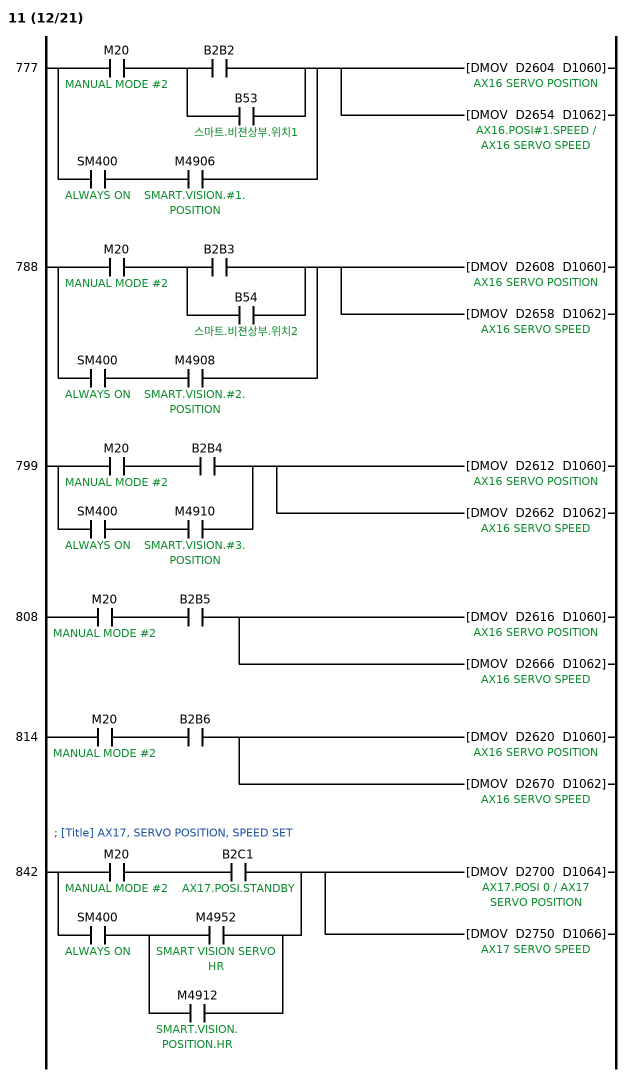
777   LD      M20  ; MANUAL MODE #2
      LD      B2B2
      OR      B53  ; 스마트.비젼상부.위치1
      ANB
      LD      SM400  ; ALWAYS ON
      AND     M4906  ; SMART.VISION.#1.POSITION
      ORB
      DMOV    D2604 D1060
      DMOV    D2654 D1062  ; AX16.POSI#1.SPEED
788   LD      M20  ; MANUAL MODE #2
      LD      B2B3
      OR      B54  ; 스마트.비젼상부.위치2
      ANB
      LD      SM400  ; ALWAYS ON
      AND     M4908  ; SMART.VISION.#2.POSITION
      ORB
      DMOV    D2608 D1060
      DMOV    D2658 D1062
799   LD      M20  ; MANUAL MODE #2
      AND     B2B4
      LD      SM400  ; ALWAYS ON
      AND     M4910  ; SMART.VISION.#3.POSITION
      ORB
      DMOV    D2612 D1060
      DMOV    D2662 D1062
808   LD      M20  ; MANUAL MODE #2
      AND     B2B5
      DMOV    D2616 D1060
      DMOV    D2666 D1062
814   LD      M20  ; MANUAL MODE #2
      AND     B2B6
      DMOV    D2620 D1060
      DMOV    D2670 D1062
; [Title] AX17, SERVO POSITION, SPEED SET
842   LD      M20  ; MANUAL MODE #2
      AND     B2C1  ; AX17.POSI.STANDBY
      LD      SM400  ; ALWAYS ON
      LD      M4952  ; SMART VISION SERVO HR
      OR      M4912  ; SMART.VISION.POSITION.HR
      ANB
      ORB
      DMOV    D2700 D1064  ; AX17.POSI 0
      DMOV    D2750 D1066
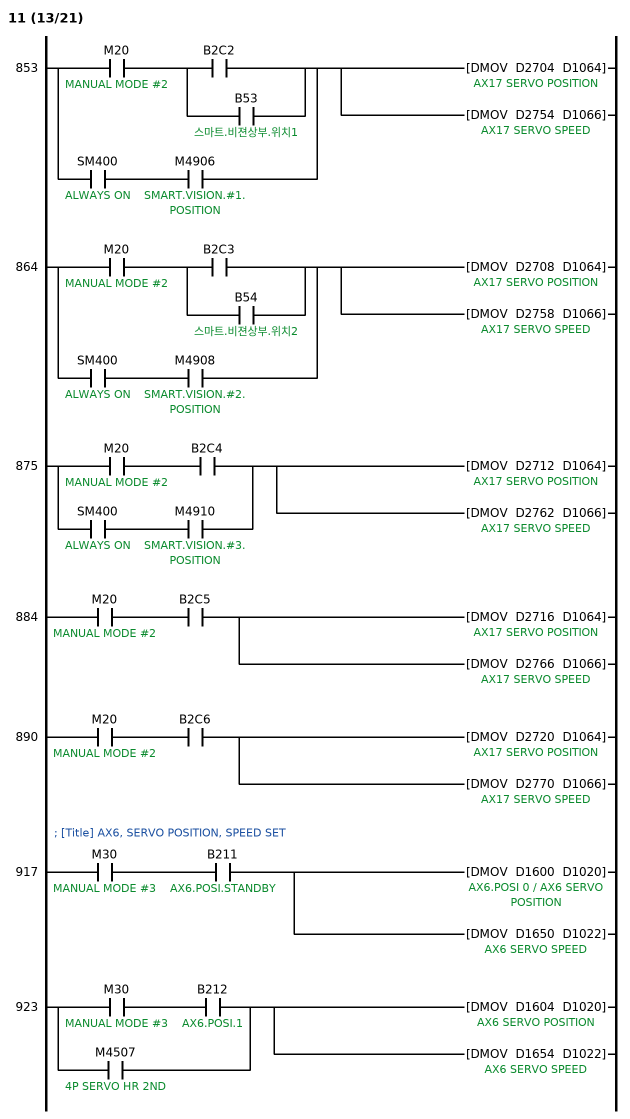
853   LD      M20  ; MANUAL MODE #2
      LD      B2C2
      OR      B53  ; 스마트.비젼상부.위치1
      ANB
      LD      SM400  ; ALWAYS ON
      AND     M4906  ; SMART.VISION.#1.POSITION
      ORB
      DMOV    D2704 D1064
      DMOV    D2754 D1066
864   LD      M20  ; MANUAL MODE #2
      LD      B2C3
      OR      B54  ; 스마트.비젼상부.위치2
      ANB
      LD      SM400  ; ALWAYS ON
      AND     M4908  ; SMART.VISION.#2.POSITION
      ORB
      DMOV    D2708 D1064
      DMOV    D2758 D1066
875   LD      M20  ; MANUAL MODE #2
      AND     B2C4
      LD      SM400  ; ALWAYS ON
      AND     M4910  ; SMART.VISION.#3.POSITION
      ORB
      DMOV    D2712 D1064
      DMOV    D2762 D1066
884   LD      M20  ; MANUAL MODE #2
      AND     B2C5
      DMOV    D2716 D1064
      DMOV    D2766 D1066
890   LD      M20  ; MANUAL MODE #2
      AND     B2C6
      DMOV    D2720 D1064
      DMOV    D2770 D1066
; [Title] AX6, SERVO POSITION, SPEED SET
917   LD      M30  ; MANUAL MODE #3
      AND     B211  ; AX6.POSI.STANDBY
      DMOV    D1600 D1020  ; AX6.POSI 0
      DMOV    D1650 D1022
923   LD      M30  ; MANUAL MODE #3
      AND     B212  ; AX6.POSI.1
      OR      M4507  ; 4P SERVO HR 2ND
      DMOV    D1604 D1020
      DMOV    D1654 D1022
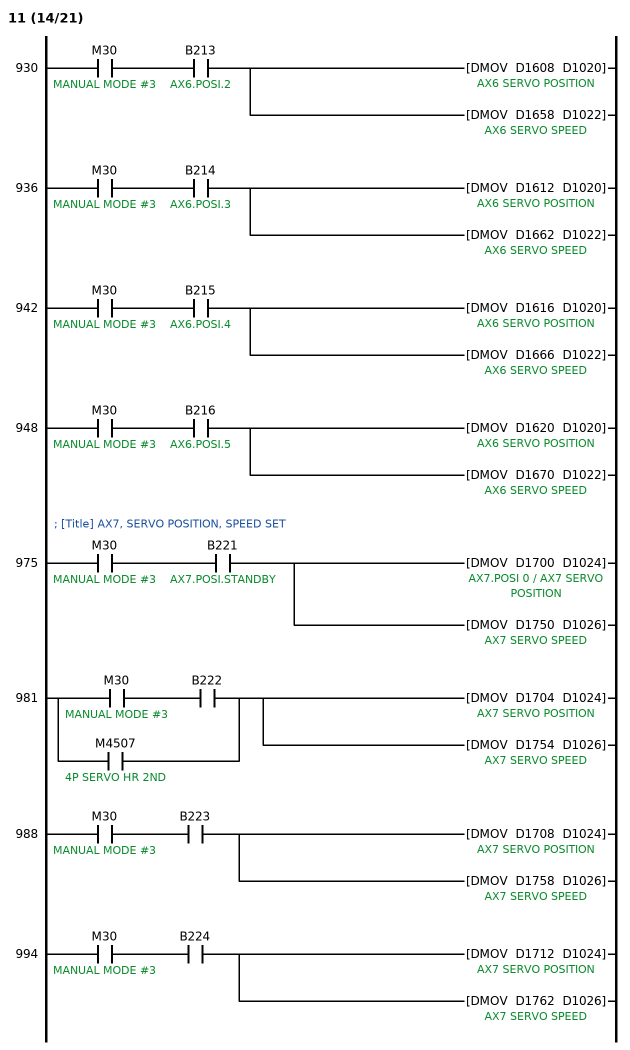
930   LD      M30  ; MANUAL MODE #3
      AND     B213  ; AX6.POSI.2
      DMOV    D1608 D1020
      DMOV    D1658 D1022
936   LD      M30  ; MANUAL MODE #3
      AND     B214  ; AX6.POSI.3
      DMOV    D1612 D1020
      DMOV    D1662 D1022
942   LD      M30  ; MANUAL MODE #3
      AND     B215  ; AX6.POSI.4
      DMOV    D1616 D1020
      DMOV    D1666 D1022
948   LD      M30  ; MANUAL MODE #3
      AND     B216  ; AX6.POSI.5
      DMOV    D1620 D1020
      DMOV    D1670 D1022
; [Title] AX7, SERVO POSITION, SPEED SET
975   LD      M30  ; MANUAL MODE #3
      AND     B221  ; AX7.POSI.STANDBY
      DMOV    D1700 D1024  ; AX7.POSI 0
      DMOV    D1750 D1026
981   LD      M30  ; MANUAL MODE #3
      AND     B222
      OR      M4507  ; 4P SERVO HR 2ND
      DMOV    D1704 D1024
      DMOV    D1754 D1026
988   LD      M30  ; MANUAL MODE #3
      AND     B223
      DMOV    D1708 D1024
      DMOV    D1758 D1026
994   LD      M30  ; MANUAL MODE #3
      AND     B224
      DMOV    D1712 D1024
      DMOV    D1762 D1026
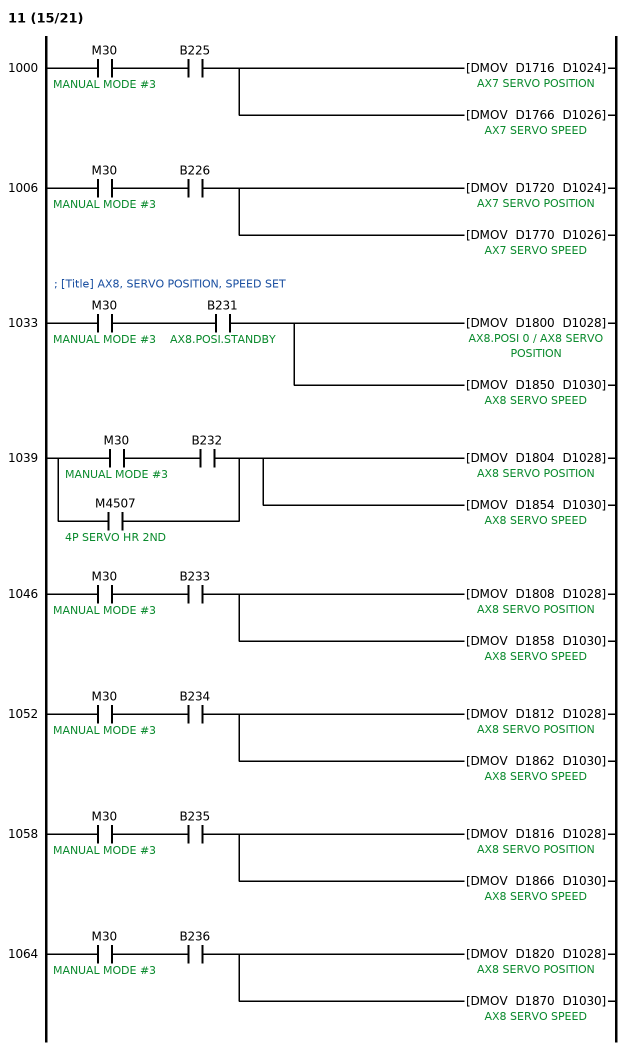
1000  LD      M30  ; MANUAL MODE #3
      AND     B225
      DMOV    D1716 D1024
      DMOV    D1766 D1026
1006  LD      M30  ; MANUAL MODE #3
      AND     B226
      DMOV    D1720 D1024
      DMOV    D1770 D1026
; [Title] AX8, SERVO POSITION, SPEED SET
1033  LD      M30  ; MANUAL MODE #3
      AND     B231  ; AX8.POSI.STANDBY
      DMOV    D1800 D1028  ; AX8.POSI 0
      DMOV    D1850 D1030
1039  LD      M30  ; MANUAL MODE #3
      AND     B232
      OR      M4507  ; 4P SERVO HR 2ND
      DMOV    D1804 D1028
      DMOV    D1854 D1030
1046  LD      M30  ; MANUAL MODE #3
      AND     B233
      DMOV    D1808 D1028
      DMOV    D1858 D1030
1052  LD      M30  ; MANUAL MODE #3
      AND     B234
      DMOV    D1812 D1028
      DMOV    D1862 D1030
1058  LD      M30  ; MANUAL MODE #3
      AND     B235
      DMOV    D1816 D1028
      DMOV    D1866 D1030
1064  LD      M30  ; MANUAL MODE #3
      AND     B236
      DMOV    D1820 D1028
      DMOV    D1870 D1030
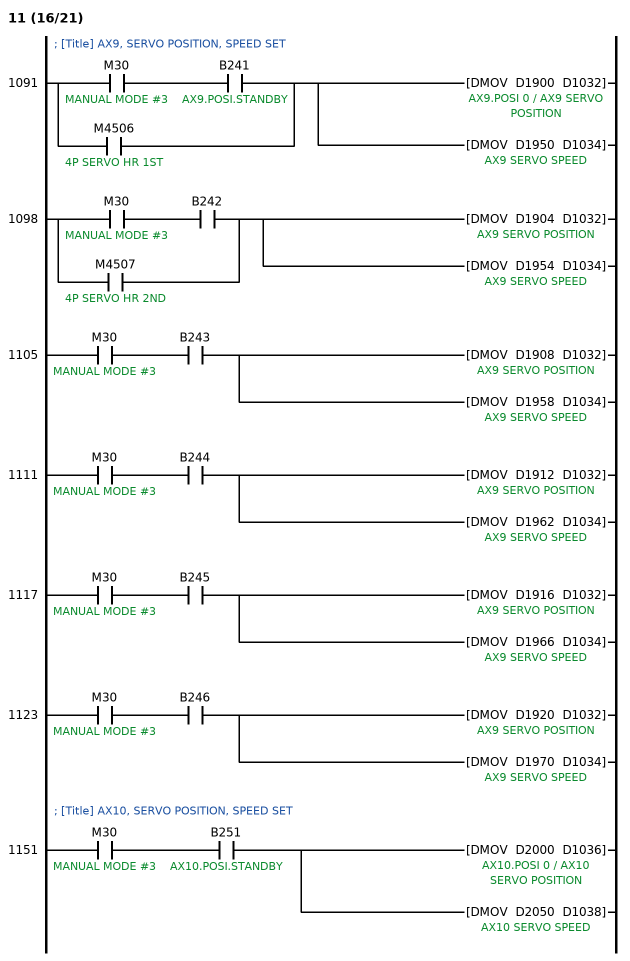
; [Title] AX9, SERVO POSITION, SPEED SET
1091  LD      M30  ; MANUAL MODE #3
      AND     B241  ; AX9.POSI.STANDBY
      OR      M4506  ; 4P SERVO HR 1ST
      DMOV    D1900 D1032  ; AX9.POSI 0
      DMOV    D1950 D1034
1098  LD      M30  ; MANUAL MODE #3
      AND     B242
      OR      M4507  ; 4P SERVO HR 2ND
      DMOV    D1904 D1032
      DMOV    D1954 D1034
1105  LD      M30  ; MANUAL MODE #3
      AND     B243
      DMOV    D1908 D1032
      DMOV    D1958 D1034
1111  LD      M30  ; MANUAL MODE #3
      AND     B244
      DMOV    D1912 D1032
      DMOV    D1962 D1034
1117  LD      M30  ; MANUAL MODE #3
      AND     B245
      DMOV    D1916 D1032
      DMOV    D1966 D1034
1123  LD      M30  ; MANUAL MODE #3
      AND     B246
      DMOV    D1920 D1032
      DMOV    D1970 D1034
; [Title] AX10, SERVO POSITION, SPEED SET
1151  LD      M30  ; MANUAL MODE #3
      AND     B251  ; AX10.POSI.STANDBY
      DMOV    D2000 D1036  ; AX10.POSI 0
      DMOV    D2050 D1038
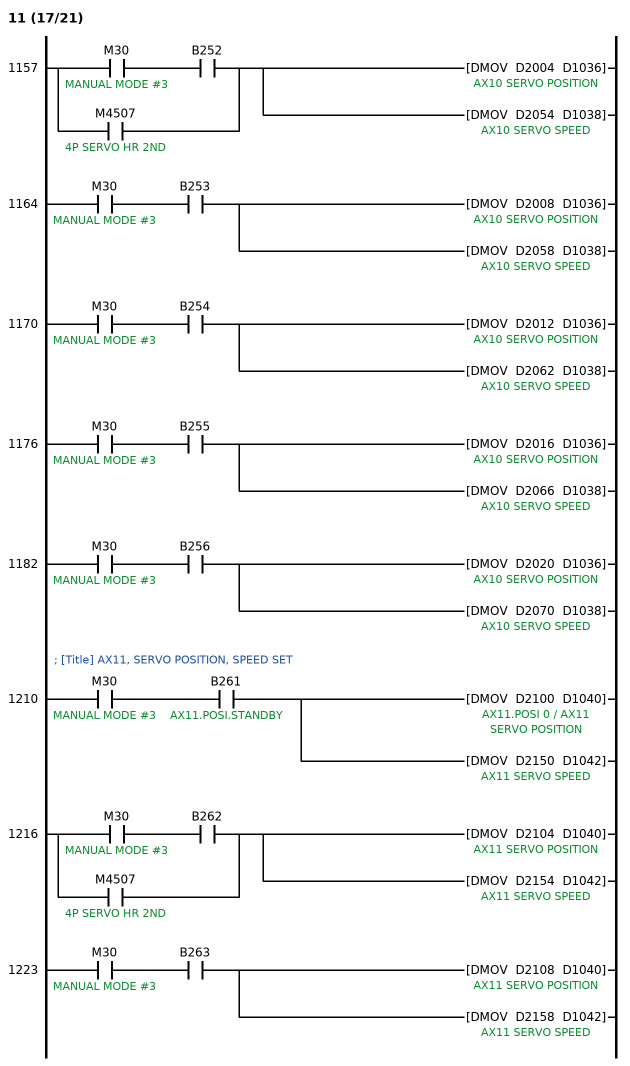
1157  LD      M30  ; MANUAL MODE #3
      AND     B252
      OR      M4507  ; 4P SERVO HR 2ND
      DMOV    D2004 D1036
      DMOV    D2054 D1038
1164  LD      M30  ; MANUAL MODE #3
      AND     B253
      DMOV    D2008 D1036
      DMOV    D2058 D1038
1170  LD      M30  ; MANUAL MODE #3
      AND     B254
      DMOV    D2012 D1036
      DMOV    D2062 D1038
1176  LD      M30  ; MANUAL MODE #3
      AND     B255
      DMOV    D2016 D1036
      DMOV    D2066 D1038
1182  LD      M30  ; MANUAL MODE #3
      AND     B256
      DMOV    D2020 D1036
      DMOV    D2070 D1038
; [Title] AX11, SERVO POSITION, SPEED SET
1210  LD      M30  ; MANUAL MODE #3
      AND     B261  ; AX11.POSI.STANDBY
      DMOV    D2100 D1040  ; AX11.POSI 0
      DMOV    D2150 D1042
1216  LD      M30  ; MANUAL MODE #3
      AND     B262
      OR      M4507  ; 4P SERVO HR 2ND
      DMOV    D2104 D1040
      DMOV    D2154 D1042
1223  LD      M30  ; MANUAL MODE #3
      AND     B263
      DMOV    D2108 D1040
      DMOV    D2158 D1042
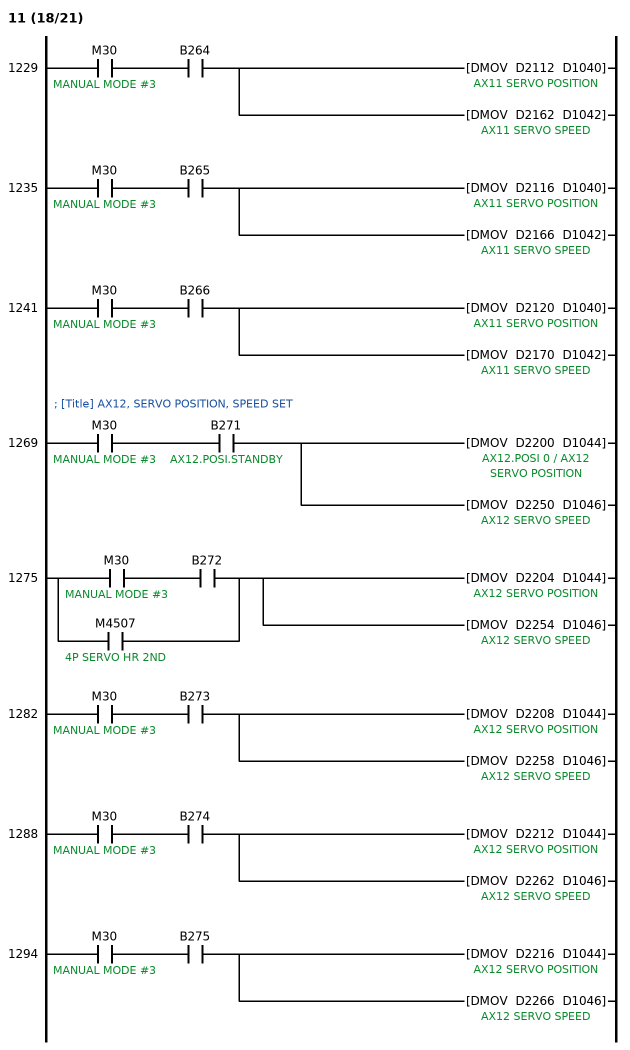
1229  LD      M30  ; MANUAL MODE #3
      AND     B264
      DMOV    D2112 D1040
      DMOV    D2162 D1042
1235  LD      M30  ; MANUAL MODE #3
      AND     B265
      DMOV    D2116 D1040
      DMOV    D2166 D1042
1241  LD      M30  ; MANUAL MODE #3
      AND     B266
      DMOV    D2120 D1040
      DMOV    D2170 D1042
; [Title] AX12, SERVO POSITION, SPEED SET
1269  LD      M30  ; MANUAL MODE #3
      AND     B271  ; AX12.POSI.STANDBY
      DMOV    D2200 D1044  ; AX12.POSI 0
      DMOV    D2250 D1046
1275  LD      M30  ; MANUAL MODE #3
      AND     B272
      OR      M4507  ; 4P SERVO HR 2ND
      DMOV    D2204 D1044
      DMOV    D2254 D1046
1282  LD      M30  ; MANUAL MODE #3
      AND     B273
      DMOV    D2208 D1044
      DMOV    D2258 D1046
1288  LD      M30  ; MANUAL MODE #3
      AND     B274
      DMOV    D2212 D1044
      DMOV    D2262 D1046
1294  LD      M30  ; MANUAL MODE #3
      AND     B275
      DMOV    D2216 D1044
      DMOV    D2266 D1046
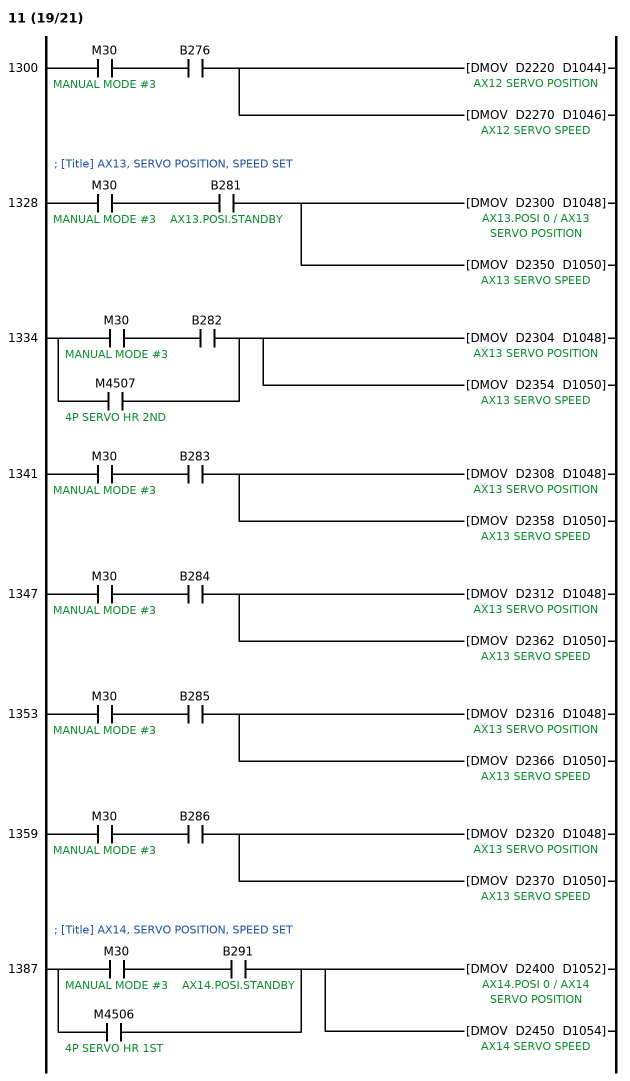
1300  LD      M30  ; MANUAL MODE #3
      AND     B276
      DMOV    D2220 D1044
      DMOV    D2270 D1046
; [Title] AX13, SERVO POSITION, SPEED SET
1328  LD      M30  ; MANUAL MODE #3
      AND     B281  ; AX13.POSI.STANDBY
      DMOV    D2300 D1048  ; AX13.POSI 0
      DMOV    D2350 D1050
1334  LD      M30  ; MANUAL MODE #3
      AND     B282
      OR      M4507  ; 4P SERVO HR 2ND
      DMOV    D2304 D1048
      DMOV    D2354 D1050
1341  LD      M30  ; MANUAL MODE #3
      AND     B283
      DMOV    D2308 D1048
      DMOV    D2358 D1050
1347  LD      M30  ; MANUAL MODE #3
      AND     B284
      DMOV    D2312 D1048
      DMOV    D2362 D1050
1353  LD      M30  ; MANUAL MODE #3
      AND     B285
      DMOV    D2316 D1048
      DMOV    D2366 D1050
1359  LD      M30  ; MANUAL MODE #3
      AND     B286
      DMOV    D2320 D1048
      DMOV    D2370 D1050
; [Title] AX14, SERVO POSITION, SPEED SET
1387  LD      M30  ; MANUAL MODE #3
      AND     B291  ; AX14.POSI.STANDBY
      OR      M4506  ; 4P SERVO HR 1ST
      DMOV    D2400 D1052  ; AX14.POSI 0
      DMOV    D2450 D1054
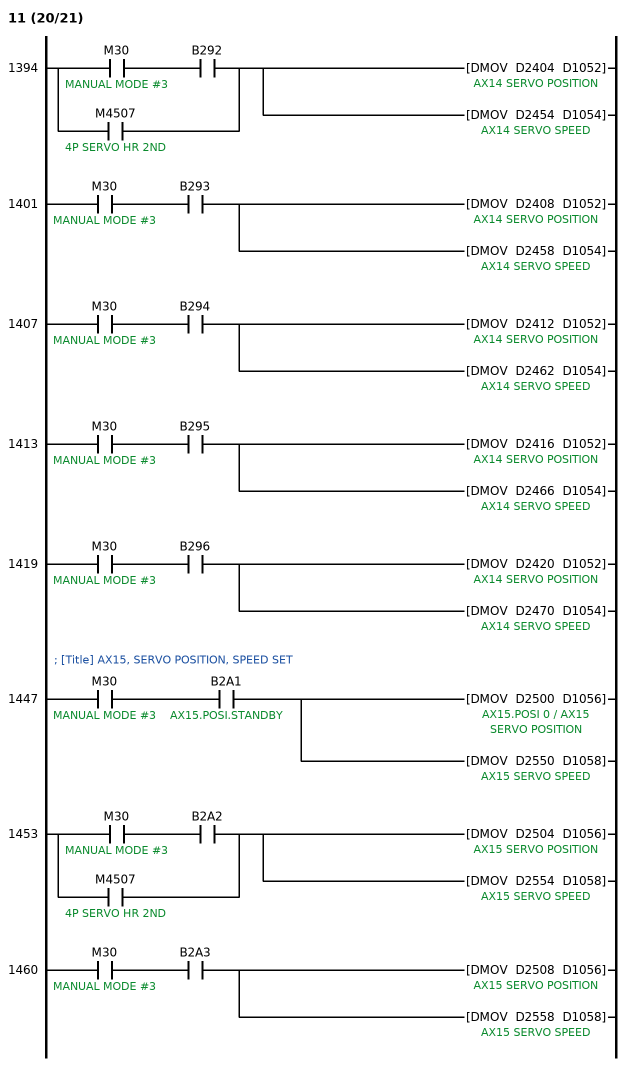
1394  LD      M30  ; MANUAL MODE #3
      AND     B292
      OR      M4507  ; 4P SERVO HR 2ND
      DMOV    D2404 D1052
      DMOV    D2454 D1054
1401  LD      M30  ; MANUAL MODE #3
      AND     B293
      DMOV    D2408 D1052
      DMOV    D2458 D1054
1407  LD      M30  ; MANUAL MODE #3
      AND     B294
      DMOV    D2412 D1052
      DMOV    D2462 D1054
1413  LD      M30  ; MANUAL MODE #3
      AND     B295
      DMOV    D2416 D1052
      DMOV    D2466 D1054
1419  LD      M30  ; MANUAL MODE #3
      AND     B296
      DMOV    D2420 D1052
      DMOV    D2470 D1054
; [Title] AX15, SERVO POSITION, SPEED SET
1447  LD      M30  ; MANUAL MODE #3
      AND     B2A1  ; AX15.POSI.STANDBY
      DMOV    D2500 D1056  ; AX15.POSI 0
      DMOV    D2550 D1058
1453  LD      M30  ; MANUAL MODE #3
      AND     B2A2
      OR      M4507  ; 4P SERVO HR 2ND
      DMOV    D2504 D1056
      DMOV    D2554 D1058
1460  LD      M30  ; MANUAL MODE #3
      AND     B2A3
      DMOV    D2508 D1056
      DMOV    D2558 D1058
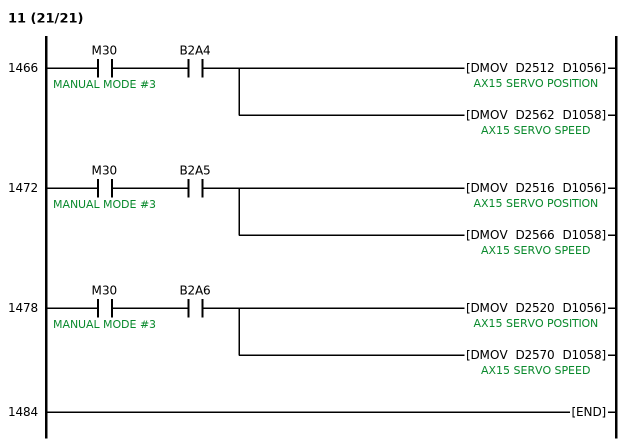
1466  LD      M30  ; MANUAL MODE #3
      AND     B2A4
      DMOV    D2512 D1056
      DMOV    D2562 D1058
1472  LD      M30  ; MANUAL MODE #3
      AND     B2A5
      DMOV    D2516 D1056
      DMOV    D2566 D1058
1478  LD      M30  ; MANUAL MODE #3
      AND     B2A6
      DMOV    D2520 D1056
      DMOV    D2570 D1058
1484  END
END_PROGRAM

PROGRAM 12  // SERVO DATA (2)
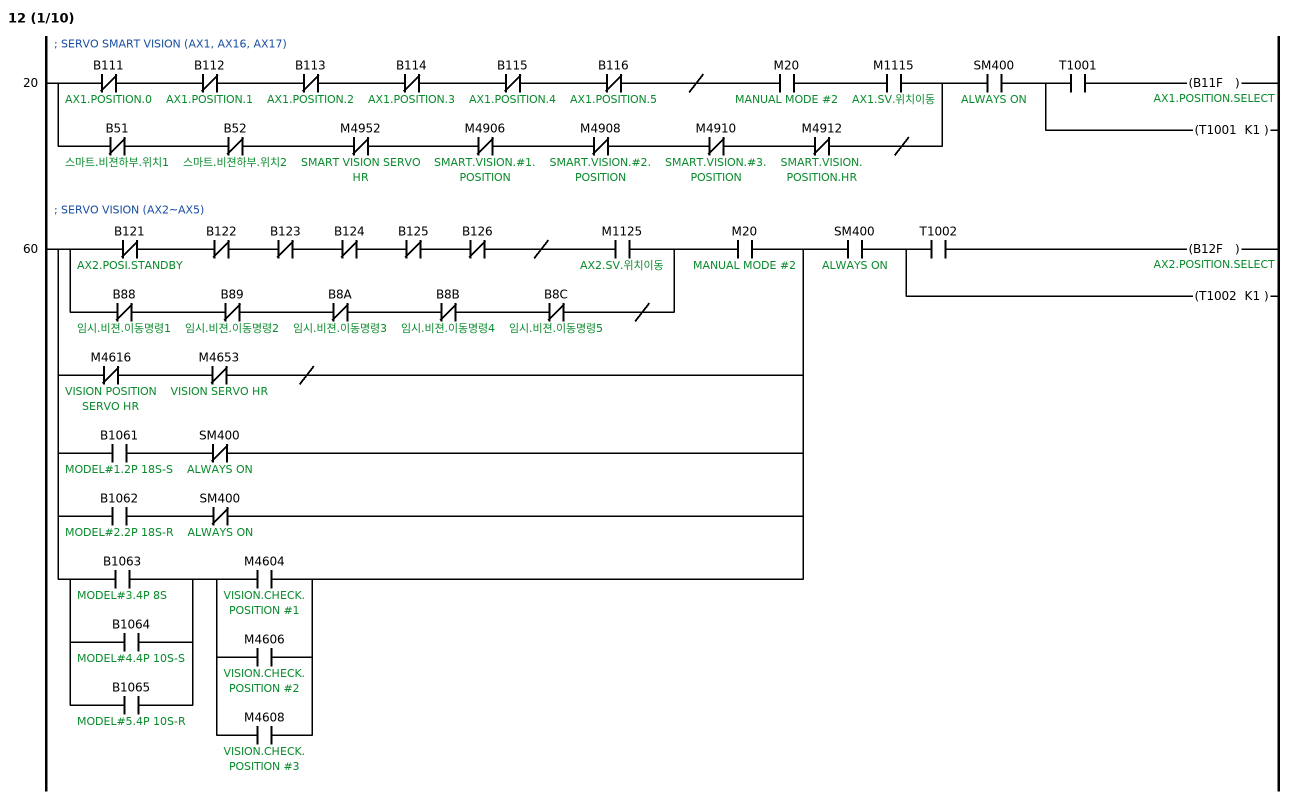
; SERVO SMART VISION (AX1, AX16, AX17)
20    LDI     B111  ; AX1.POSITION.0
      ANI     B112  ; AX1.POSITION.1
      ANI     B113  ; AX1.POSITION.2
      ANI     B114  ; AX1.POSITION.3
      ANI     B115  ; AX1.POSITION.4
      ANI     B116  ; AX1.POSITION.5
      INV
      AND     M20  ; MANUAL MODE #2
      AND     M1115  ; AX1.SV.위치이동
      LDI     B51  ; 스마트.비젼하부.위치1
      ANI     B52  ; 스마트.비젼하부.위치2
      ANI     M4952  ; SMART VISION SERVO HR
      ANI     M4906  ; SMART.VISION.#1.POSITION
      ANI     M4908  ; SMART.VISION.#2.POSITION
      ANI     M4910  ; SMART.VISION.#3.POSITION
      ANI     M4912  ; SMART.VISION.POSITION.HR
      INV
      ORB
      AND     SM400  ; ALWAYS ON
      MPS
      AND     T1001
      OUT     B11F  ; AX1.POSITION.SELECT
      MPP
      OUT     T1001 K1
; SERVO VISION (AX2~AX5)
60    LDI     B121  ; AX2.POSI.STANDBY
      ANI     B122
      ANI     B123
      ANI     B124
      ANI     B125
      ANI     B126
      INV
      AND     M1125  ; AX2.SV.위치이동
      LDI     B88  ; 임시.비젼.이동명령1
      ANI     B89  ; 임시.비젼.이동명령2
      ANI     B8A  ; 임시.비젼.이동명령3
      ANI     B8B  ; 임시.비젼.이동명령4
      ANI     B8C  ; 임시.비젼.이동명령5
      INV
      ORB
      AND     M20  ; MANUAL MODE #2
      LDI     M4616  ; VISION POSITION SERVO HR
      ANI     M4653  ; VISION SERVO HR
      INV
      ORB
      LD      B1061  ; MODEL#1.2P 18S-S
      ANI     SM400  ; ALWAYS ON
      ORB
      LD      B1062  ; MODEL#2.2P 18S-R
      ANI     SM400  ; ALWAYS ON
      ORB
      LD      B1063  ; MODEL#3.4P 8S
      OR      B1064  ; MODEL#4.4P 10S-S
      OR      B1065  ; MODEL#5.4P 10S-R
      LD      M4604  ; VISION.CHECK.POSITION #1
      OR      M4606  ; VISION.CHECK.POSITION #2
      OR      M4608  ; VISION.CHECK.POSITION #3
      ANB
      ORB
      AND     SM400  ; ALWAYS ON
      MPS
      AND     T1002
      OUT     B12F  ; AX2.POSITION.SELECT
      MPP
      OUT     T1002 K1
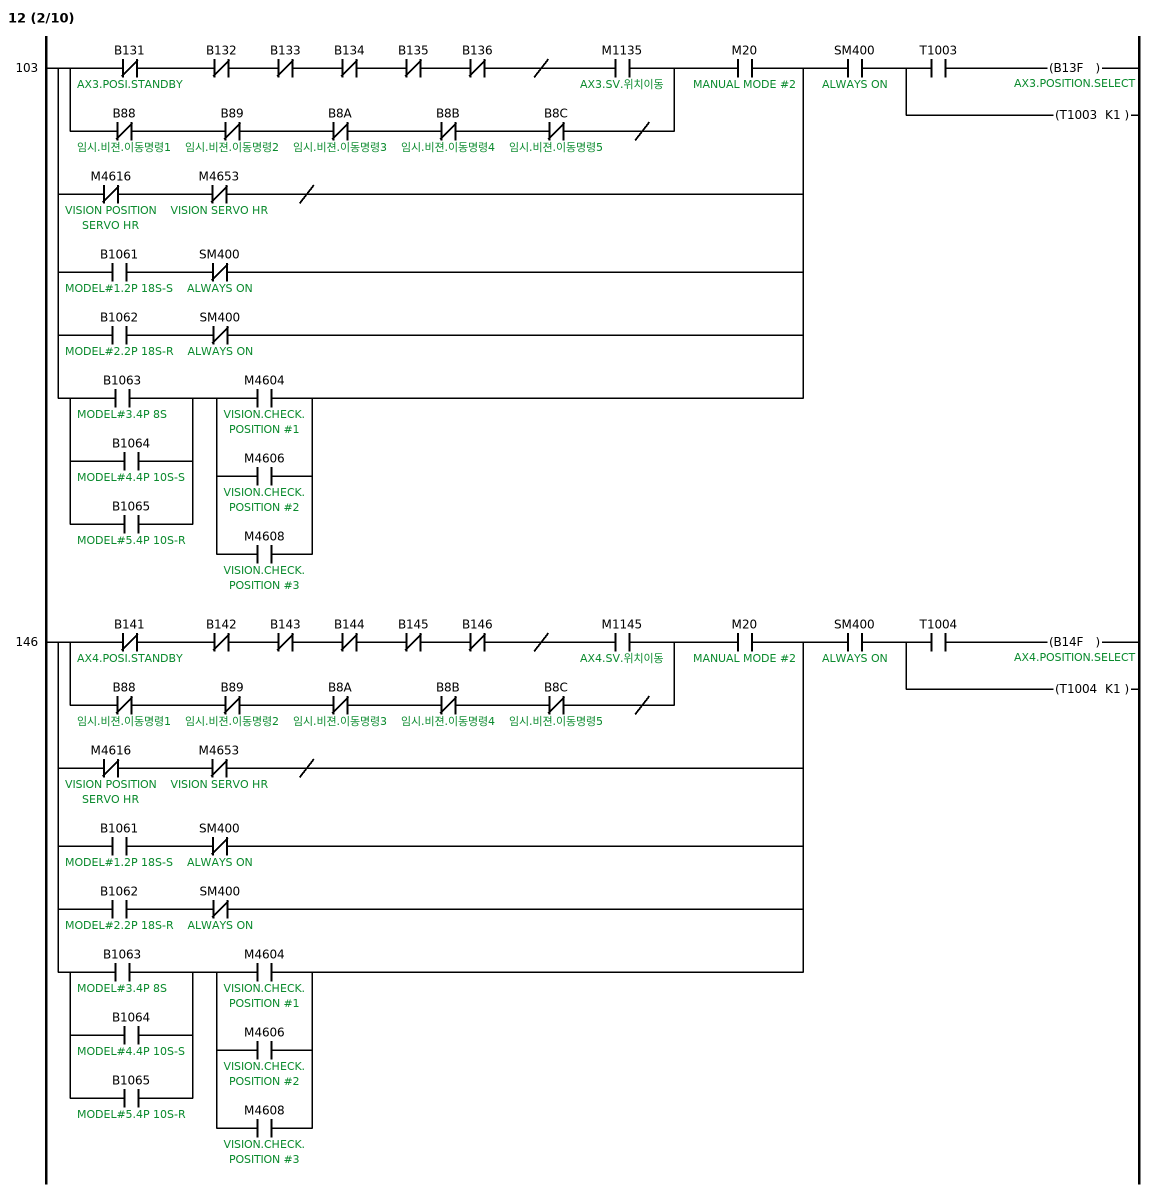
103   LDI     B131  ; AX3.POSI.STANDBY
      ANI     B132
      ANI     B133
      ANI     B134
      ANI     B135
      ANI     B136
      INV
      AND     M1135  ; AX3.SV.위치이동
      LDI     B88  ; 임시.비젼.이동명령1
      ANI     B89  ; 임시.비젼.이동명령2
      ANI     B8A  ; 임시.비젼.이동명령3
      ANI     B8B  ; 임시.비젼.이동명령4
      ANI     B8C  ; 임시.비젼.이동명령5
      INV
      ORB
      AND     M20  ; MANUAL MODE #2
      LDI     M4616  ; VISION POSITION SERVO HR
      ANI     M4653  ; VISION SERVO HR
      INV
      ORB
      LD      B1061  ; MODEL#1.2P 18S-S
      ANI     SM400  ; ALWAYS ON
      ORB
      LD      B1062  ; MODEL#2.2P 18S-R
      ANI     SM400  ; ALWAYS ON
      ORB
      LD      B1063  ; MODEL#3.4P 8S
      OR      B1064  ; MODEL#4.4P 10S-S
      OR      B1065  ; MODEL#5.4P 10S-R
      LD      M4604  ; VISION.CHECK.POSITION #1
      OR      M4606  ; VISION.CHECK.POSITION #2
      OR      M4608  ; VISION.CHECK.POSITION #3
      ANB
      ORB
      AND     SM400  ; ALWAYS ON
      MPS
      AND     T1003
      OUT     B13F  ; AX3.POSITION.SELECT
      MPP
      OUT     T1003 K1
146   LDI     B141  ; AX4.POSI.STANDBY
      ANI     B142
      ANI     B143
      ANI     B144
      ANI     B145
      ANI     B146
      INV
      AND     M1145  ; AX4.SV.위치이동
      LDI     B88  ; 임시.비젼.이동명령1
      ANI     B89  ; 임시.비젼.이동명령2
      ANI     B8A  ; 임시.비젼.이동명령3
      ANI     B8B  ; 임시.비젼.이동명령4
      ANI     B8C  ; 임시.비젼.이동명령5
      INV
      ORB
      AND     M20  ; MANUAL MODE #2
      LDI     M4616  ; VISION POSITION SERVO HR
      ANI     M4653  ; VISION SERVO HR
      INV
      ORB
      LD      B1061  ; MODEL#1.2P 18S-S
      ANI     SM400  ; ALWAYS ON
      ORB
      LD      B1062  ; MODEL#2.2P 18S-R
      ANI     SM400  ; ALWAYS ON
      ORB
      LD      B1063  ; MODEL#3.4P 8S
      OR      B1064  ; MODEL#4.4P 10S-S
      OR      B1065  ; MODEL#5.4P 10S-R
      LD      M4604  ; VISION.CHECK.POSITION #1
      OR      M4606  ; VISION.CHECK.POSITION #2
      OR      M4608  ; VISION.CHECK.POSITION #3
      ANB
      ORB
      AND     SM400  ; ALWAYS ON
      MPS
      AND     T1004
      OUT     B14F  ; AX4.POSITION.SELECT
      MPP
      OUT     T1004 K1
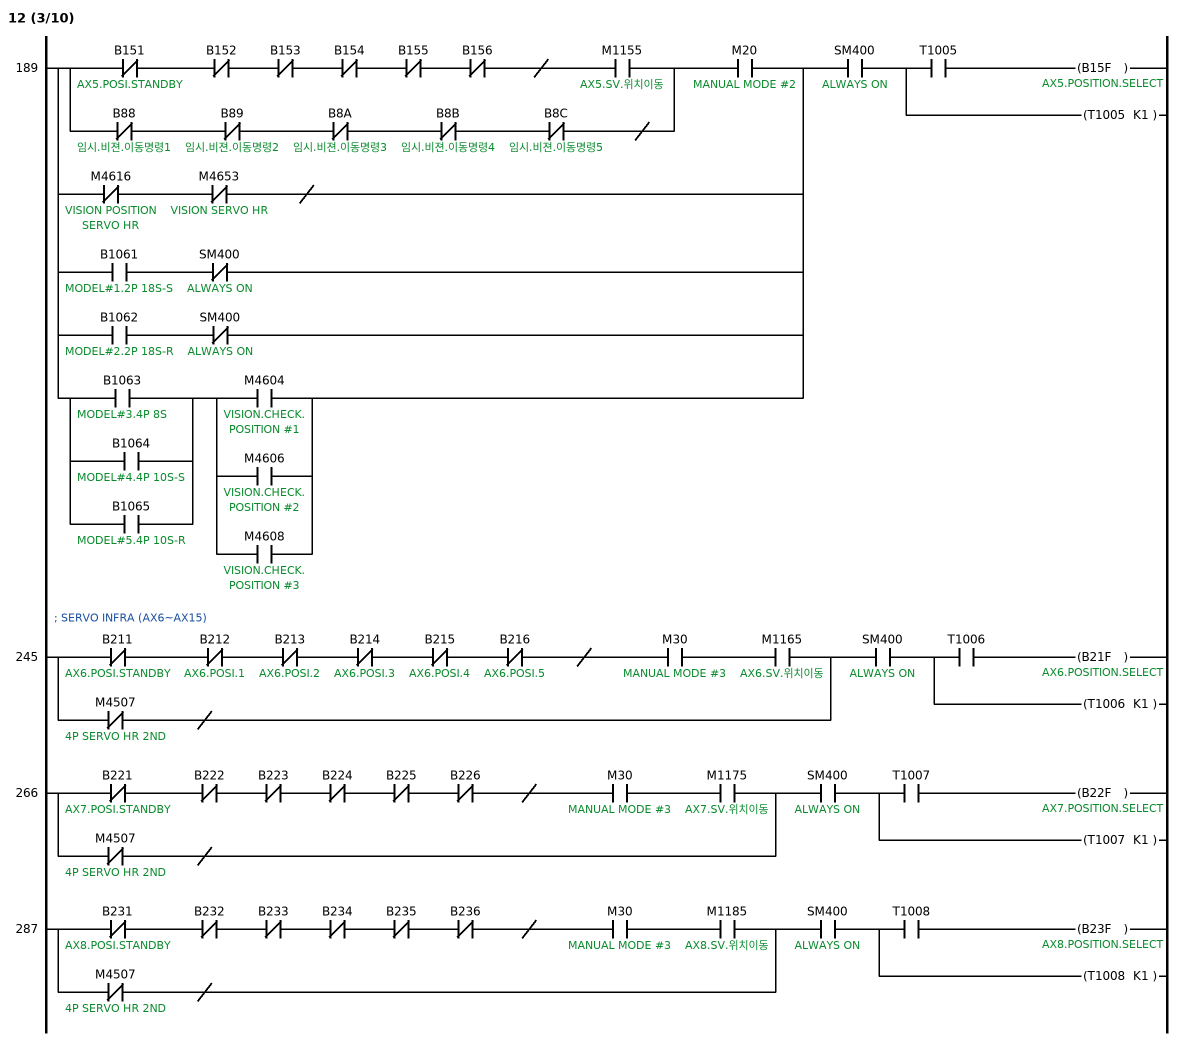
189   LDI     B151  ; AX5.POSI.STANDBY
      ANI     B152
      ANI     B153
      ANI     B154
      ANI     B155
      ANI     B156
      INV
      AND     M1155  ; AX5.SV.위치이동
      LDI     B88  ; 임시.비젼.이동명령1
      ANI     B89  ; 임시.비젼.이동명령2
      ANI     B8A  ; 임시.비젼.이동명령3
      ANI     B8B  ; 임시.비젼.이동명령4
      ANI     B8C  ; 임시.비젼.이동명령5
      INV
      ORB
      AND     M20  ; MANUAL MODE #2
      LDI     M4616  ; VISION POSITION SERVO HR
      ANI     M4653  ; VISION SERVO HR
      INV
      ORB
      LD      B1061  ; MODEL#1.2P 18S-S
      ANI     SM400  ; ALWAYS ON
      ORB
      LD      B1062  ; MODEL#2.2P 18S-R
      ANI     SM400  ; ALWAYS ON
      ORB
      LD      B1063  ; MODEL#3.4P 8S
      OR      B1064  ; MODEL#4.4P 10S-S
      OR      B1065  ; MODEL#5.4P 10S-R
      LD      M4604  ; VISION.CHECK.POSITION #1
      OR      M4606  ; VISION.CHECK.POSITION #2
      OR      M4608  ; VISION.CHECK.POSITION #3
      ANB
      ORB
      AND     SM400  ; ALWAYS ON
      MPS
      AND     T1005
      OUT     B15F  ; AX5.POSITION.SELECT
      MPP
      OUT     T1005 K1
; SERVO INFRA (AX6~AX15)
245   LDI     B211  ; AX6.POSI.STANDBY
      ANI     B212  ; AX6.POSI.1
      ANI     B213  ; AX6.POSI.2
      ANI     B214  ; AX6.POSI.3
      ANI     B215  ; AX6.POSI.4
      ANI     B216  ; AX6.POSI.5
      INV
      AND     M30  ; MANUAL MODE #3
      AND     M1165  ; AX6.SV.위치이동
      LDI     M4507  ; 4P SERVO HR 2ND
      INV
      ORB
      AND     SM400  ; ALWAYS ON
      MPS
      AND     T1006
      OUT     B21F  ; AX6.POSITION.SELECT
      MPP
      OUT     T1006 K1
266   LDI     B221  ; AX7.POSI.STANDBY
      ANI     B222
      ANI     B223
      ANI     B224
      ANI     B225
      ANI     B226
      INV
      AND     M30  ; MANUAL MODE #3
      AND     M1175  ; AX7.SV.위치이동
      LDI     M4507  ; 4P SERVO HR 2ND
      INV
      ORB
      AND     SM400  ; ALWAYS ON
      MPS
      AND     T1007
      OUT     B22F  ; AX7.POSITION.SELECT
      MPP
      OUT     T1007 K1
287   LDI     B231  ; AX8.POSI.STANDBY
      ANI     B232
      ANI     B233
      ANI     B234
      ANI     B235
      ANI     B236
      INV
      AND     M30  ; MANUAL MODE #3
      AND     M1185  ; AX8.SV.위치이동
      LDI     M4507  ; 4P SERVO HR 2ND
      INV
      ORB
      AND     SM400  ; ALWAYS ON
      MPS
      AND     T1008
      OUT     B23F  ; AX8.POSITION.SELECT
      MPP
      OUT     T1008 K1
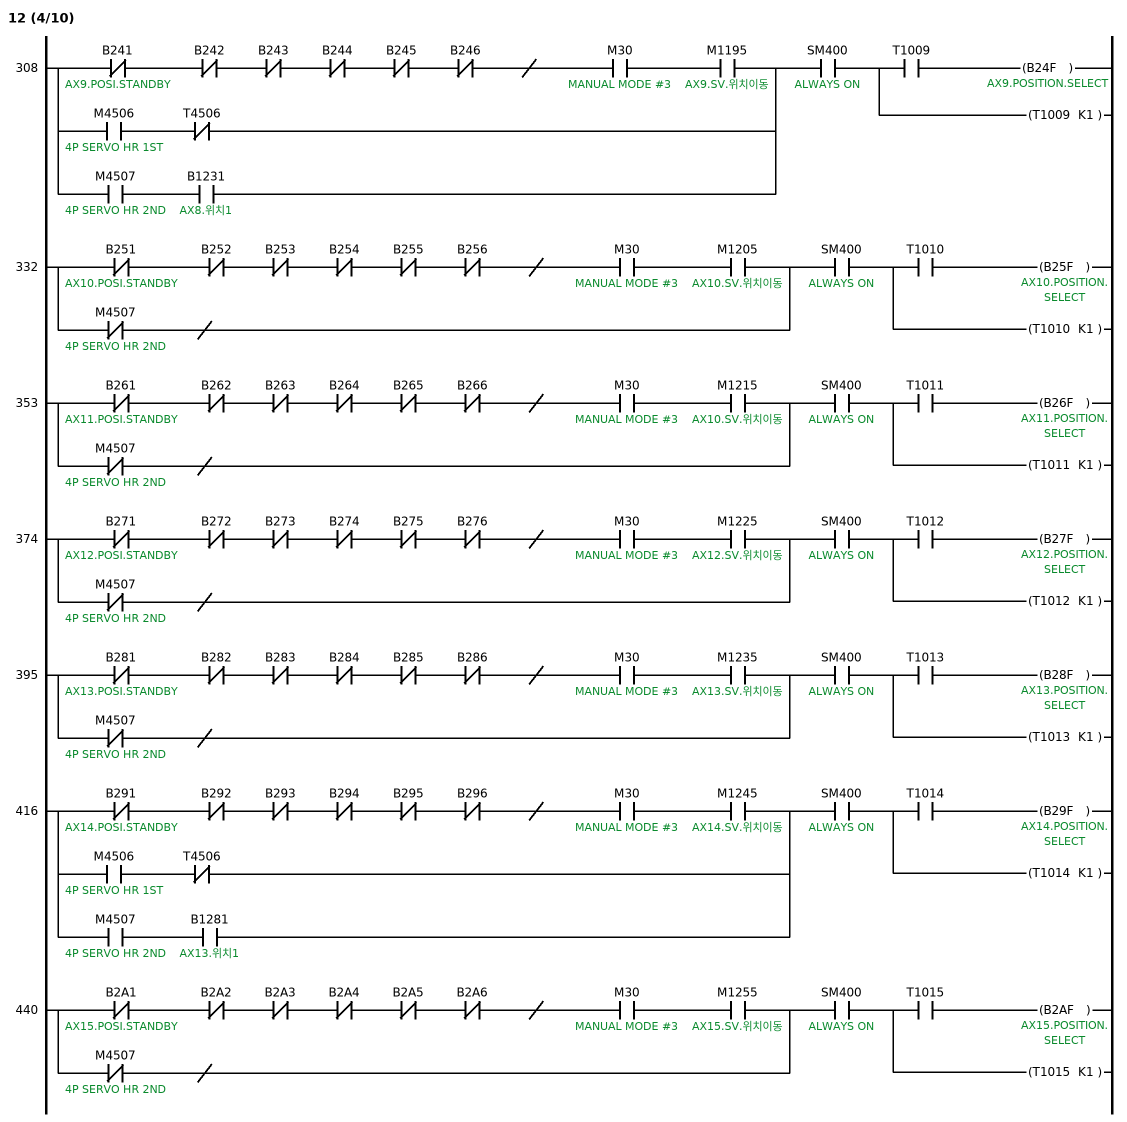
308   LDI     B241  ; AX9.POSI.STANDBY
      ANI     B242
      ANI     B243
      ANI     B244
      ANI     B245
      ANI     B246
      INV
      AND     M30  ; MANUAL MODE #3
      AND     M1195  ; AX9.SV.위치이동
      LD      M4506  ; 4P SERVO HR 1ST
      ANI     T4506
      ORB
      LD      M4507  ; 4P SERVO HR 2ND
      AND     B1231  ; AX8.위치1
      ORB
      AND     SM400  ; ALWAYS ON
      MPS
      AND     T1009
      OUT     B24F  ; AX9.POSITION.SELECT
      MPP
      OUT     T1009 K1
332   LDI     B251  ; AX10.POSI.STANDBY
      ANI     B252
      ANI     B253
      ANI     B254
      ANI     B255
      ANI     B256
      INV
      AND     M30  ; MANUAL MODE #3
      AND     M1205  ; AX10.SV.위치이동
      LDI     M4507  ; 4P SERVO HR 2ND
      INV
      ORB
      AND     SM400  ; ALWAYS ON
      MPS
      AND     T1010
      OUT     B25F  ; AX10.POSITION.SELECT
      MPP
      OUT     T1010 K1
353   LDI     B261  ; AX11.POSI.STANDBY
      ANI     B262
      ANI     B263
      ANI     B264
      ANI     B265
      ANI     B266
      INV
      AND     M30  ; MANUAL MODE #3
      AND     M1215  ; AX10.SV.위치이동
      LDI     M4507  ; 4P SERVO HR 2ND
      INV
      ORB
      AND     SM400  ; ALWAYS ON
      MPS
      AND     T1011
      OUT     B26F  ; AX11.POSITION.SELECT
      MPP
      OUT     T1011 K1
374   LDI     B271  ; AX12.POSI.STANDBY
      ANI     B272
      ANI     B273
      ANI     B274
      ANI     B275
      ANI     B276
      INV
      AND     M30  ; MANUAL MODE #3
      AND     M1225  ; AX12.SV.위치이동
      LDI     M4507  ; 4P SERVO HR 2ND
      INV
      ORB
      AND     SM400  ; ALWAYS ON
      MPS
      AND     T1012
      OUT     B27F  ; AX12.POSITION.SELECT
      MPP
      OUT     T1012 K1
395   LDI     B281  ; AX13.POSI.STANDBY
      ANI     B282
      ANI     B283
      ANI     B284
      ANI     B285
      ANI     B286
      INV
      AND     M30  ; MANUAL MODE #3
      AND     M1235  ; AX13.SV.위치이동
      LDI     M4507  ; 4P SERVO HR 2ND
      INV
      ORB
      AND     SM400  ; ALWAYS ON
      MPS
      AND     T1013
      OUT     B28F  ; AX13.POSITION.SELECT
      MPP
      OUT     T1013 K1
416   LDI     B291  ; AX14.POSI.STANDBY
      ANI     B292
      ANI     B293
      ANI     B294
      ANI     B295
      ANI     B296
      INV
      AND     M30  ; MANUAL MODE #3
      AND     M1245  ; AX14.SV.위치이동
      LD      M4506  ; 4P SERVO HR 1ST
      ANI     T4506
      ORB
      LD      M4507  ; 4P SERVO HR 2ND
      AND     B1281  ; AX13.위치1
      ORB
      AND     SM400  ; ALWAYS ON
      MPS
      AND     T1014
      OUT     B29F  ; AX14.POSITION.SELECT
      MPP
      OUT     T1014 K1
440   LDI     B2A1  ; AX15.POSI.STANDBY
      ANI     B2A2
      ANI     B2A3
      ANI     B2A4
      ANI     B2A5
      ANI     B2A6
      INV
      AND     M30  ; MANUAL MODE #3
      AND     M1255  ; AX15.SV.위치이동
      LDI     M4507  ; 4P SERVO HR 2ND
      INV
      ORB
      AND     SM400  ; ALWAYS ON
      MPS
      AND     T1015
      OUT     B2AF  ; AX15.POSITION.SELECT
      MPP
      OUT     T1015 K1
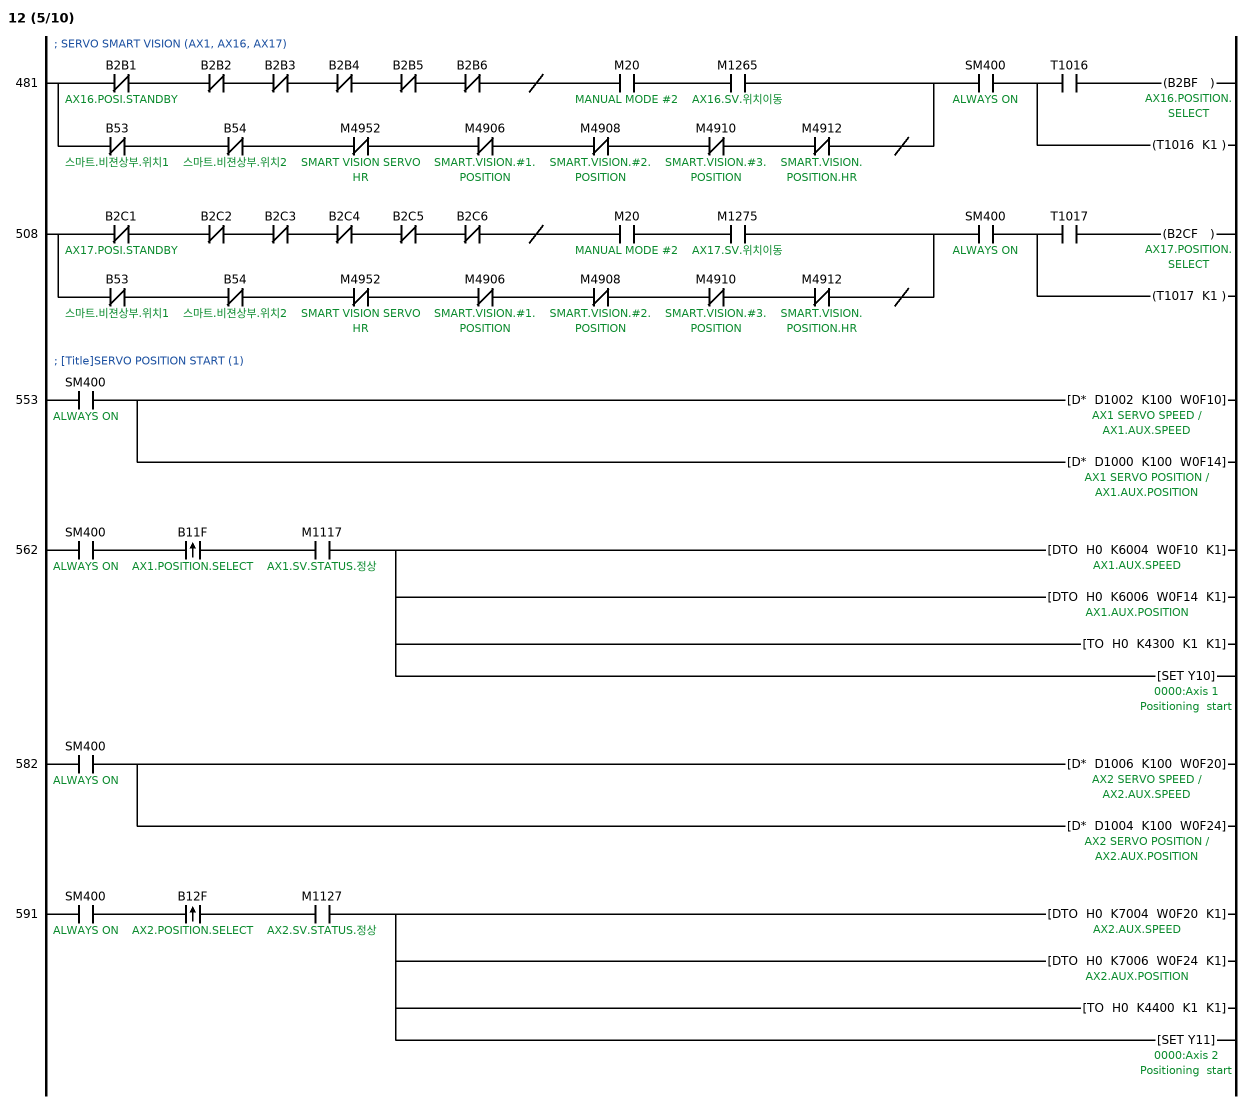
; SERVO SMART VISION (AX1, AX16, AX17)
481   LDI     B2B1  ; AX16.POSI.STANDBY
      ANI     B2B2
      ANI     B2B3
      ANI     B2B4
      ANI     B2B5
      ANI     B2B6
      INV
      AND     M20  ; MANUAL MODE #2
      AND     M1265  ; AX16.SV.위치이동
      LDI     B53  ; 스마트.비젼상부.위치1
      ANI     B54  ; 스마트.비젼상부.위치2
      ANI     M4952  ; SMART VISION SERVO HR
      ANI     M4906  ; SMART.VISION.#1.POSITION
      ANI     M4908  ; SMART.VISION.#2.POSITION
      ANI     M4910  ; SMART.VISION.#3.POSITION
      ANI     M4912  ; SMART.VISION.POSITION.HR
      INV
      ORB
      AND     SM400  ; ALWAYS ON
      MPS
      AND     T1016
      OUT     B2BF  ; AX16.POSITION.SELECT
      MPP
      OUT     T1016 K1
508   LDI     B2C1  ; AX17.POSI.STANDBY
      ANI     B2C2
      ANI     B2C3
      ANI     B2C4
      ANI     B2C5
      ANI     B2C6
      INV
      AND     M20  ; MANUAL MODE #2
      AND     M1275  ; AX17.SV.위치이동
      LDI     B53  ; 스마트.비젼상부.위치1
      ANI     B54  ; 스마트.비젼상부.위치2
      ANI     M4952  ; SMART VISION SERVO HR
      ANI     M4906  ; SMART.VISION.#1.POSITION
      ANI     M4908  ; SMART.VISION.#2.POSITION
      ANI     M4910  ; SMART.VISION.#3.POSITION
      ANI     M4912  ; SMART.VISION.POSITION.HR
      INV
      ORB
      AND     SM400  ; ALWAYS ON
      MPS
      AND     T1017
      OUT     B2CF  ; AX17.POSITION.SELECT
      MPP
      OUT     T1017 K1
; [Title]SERVO POSITION START (1)
553   LD      SM400  ; ALWAYS ON
      D*      D1002 K100 W0F10  ; AX1 SERVO SPEED / AX1.AUX.SPEED
      D*      D1000 K100 W0F14  ; AX1 SERVO POSITION / AX1.AUX.POSITION
562   LD      SM400  ; ALWAYS ON
      ANDP    B11F  ; AX1.POSITION.SELECT
      AND     M1117  ; AX1.SV.STATUS.정상
      DTO     H0 K6004 W0F10 K1
      DTO     H0 K6006 W0F14 K1
      TO      H0 K4300 K1 K1
      SET     Y10  ; 0000:Axis 1  Positioning  start
582   LD      SM400  ; ALWAYS ON
      D*      D1006 K100 W0F20  ; AX2 SERVO SPEED / AX2.AUX.SPEED
      D*      D1004 K100 W0F24  ; AX2 SERVO POSITION / AX2.AUX.POSITION
591   LD      SM400  ; ALWAYS ON
      ANDP    B12F  ; AX2.POSITION.SELECT
      AND     M1127  ; AX2.SV.STATUS.정상
      DTO     H0 K7004 W0F20 K1
      DTO     H0 K7006 W0F24 K1
      TO      H0 K4400 K1 K1
      SET     Y11  ; 0000:Axis 2  Positioning  start
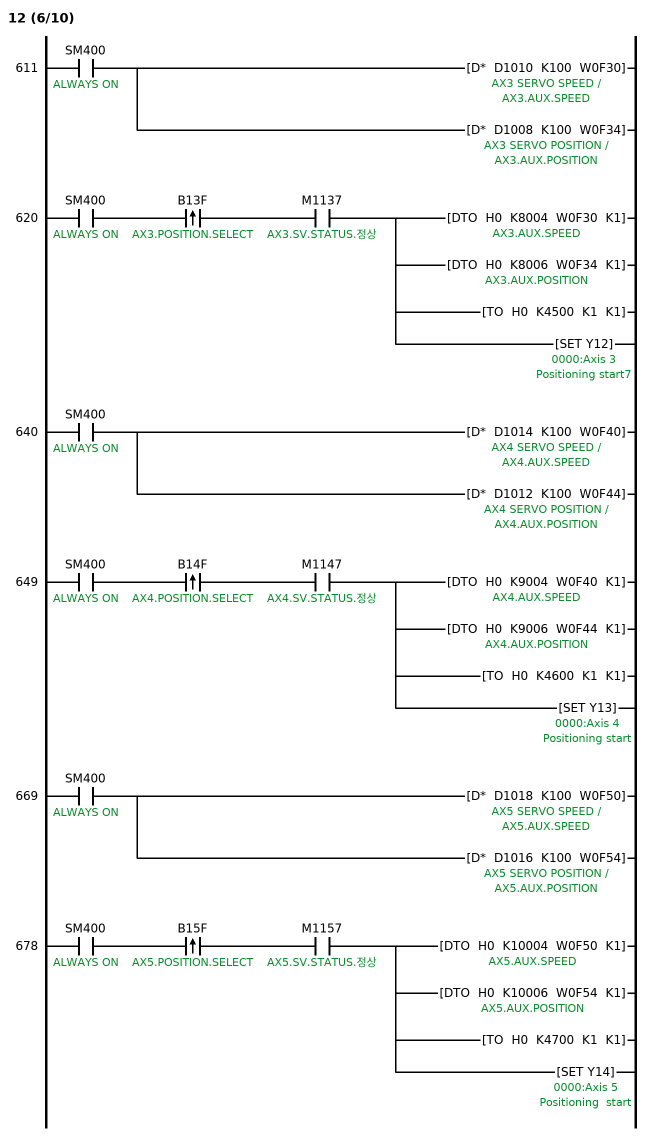
611   LD      SM400  ; ALWAYS ON
      D*      D1010 K100 W0F30  ; AX3 SERVO SPEED / AX3.AUX.SPEED
      D*      D1008 K100 W0F34  ; AX3 SERVO POSITION / AX3.AUX.POSITION
620   LD      SM400  ; ALWAYS ON
      ANDP    B13F  ; AX3.POSITION.SELECT
      AND     M1137  ; AX3.SV.STATUS.정상
      DTO     H0 K8004 W0F30 K1
      DTO     H0 K8006 W0F34 K1
      TO      H0 K4500 K1 K1
      SET     Y12  ; 0000:Axis 3 Positioning start7
640   LD      SM400  ; ALWAYS ON
      D*      D1014 K100 W0F40  ; AX4 SERVO SPEED / AX4.AUX.SPEED
      D*      D1012 K100 W0F44  ; AX4 SERVO POSITION / AX4.AUX.POSITION
649   LD      SM400  ; ALWAYS ON
      ANDP    B14F  ; AX4.POSITION.SELECT
      AND     M1147  ; AX4.SV.STATUS.정상
      DTO     H0 K9004 W0F40 K1
      DTO     H0 K9006 W0F44 K1
      TO      H0 K4600 K1 K1
      SET     Y13  ; 0000:Axis 4 Positioning start
669   LD      SM400  ; ALWAYS ON
      D*      D1018 K100 W0F50  ; AX5 SERVO SPEED / AX5.AUX.SPEED
      D*      D1016 K100 W0F54  ; AX5 SERVO POSITION / AX5.AUX.POSITION
678   LD      SM400  ; ALWAYS ON
      ANDP    B15F  ; AX5.POSITION.SELECT
      AND     M1157  ; AX5.SV.STATUS.정상
      DTO     H0 K10004 W0F50 K1
      DTO     H0 K10006 W0F54 K1
      TO      H0 K4700 K1 K1
      SET     Y14  ; 0000:Axis 5  Positioning  start
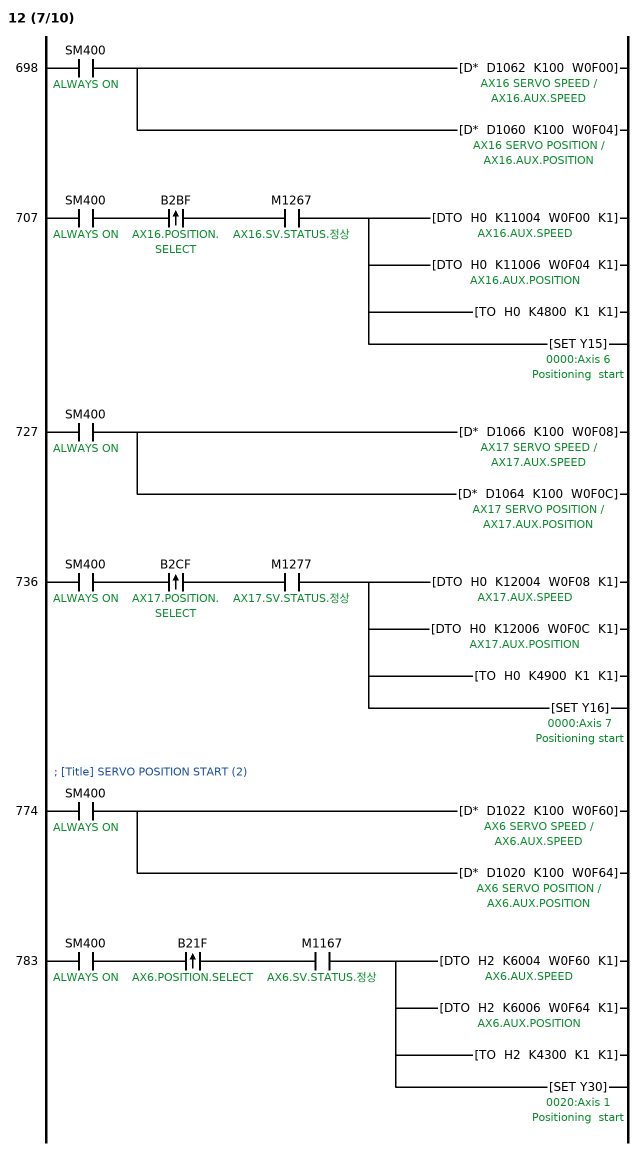
698   LD      SM400  ; ALWAYS ON
      D*      D1062 K100 W0F00  ; AX16 SERVO SPEED / AX16.AUX.SPEED
      D*      D1060 K100 W0F04  ; AX16 SERVO POSITION / AX16.AUX.POSITION
707   LD      SM400  ; ALWAYS ON
      ANDP    B2BF  ; AX16.POSITION.SELECT
      AND     M1267  ; AX16.SV.STATUS.정상
      DTO     H0 K11004 W0F00 K1
      DTO     H0 K11006 W0F04 K1
      TO      H0 K4800 K1 K1
      SET     Y15  ; 0000:Axis 6  Positioning  start
727   LD      SM400  ; ALWAYS ON
      D*      D1066 K100 W0F08  ; AX17 SERVO SPEED / AX17.AUX.SPEED
      D*      D1064 K100 W0F0C  ; AX17 SERVO POSITION / AX17.AUX.POSITION
736   LD      SM400  ; ALWAYS ON
      ANDP    B2CF  ; AX17.POSITION.SELECT
      AND     M1277  ; AX17.SV.STATUS.정상
      DTO     H0 K12004 W0F08 K1
      DTO     H0 K12006 W0F0C K1
      TO      H0 K4900 K1 K1
      SET     Y16  ; 0000:Axis 7 Positioning start
; [Title] SERVO POSITION START (2)
774   LD      SM400  ; ALWAYS ON
      D*      D1022 K100 W0F60  ; AX6 SERVO SPEED / AX6.AUX.SPEED
      D*      D1020 K100 W0F64  ; AX6 SERVO POSITION / AX6.AUX.POSITION
783   LD      SM400  ; ALWAYS ON
      ANDP    B21F  ; AX6.POSITION.SELECT
      AND     M1167  ; AX6.SV.STATUS.정상
      DTO     H2 K6004 W0F60 K1
      DTO     H2 K6006 W0F64 K1
      TO      H2 K4300 K1 K1
      SET     Y30  ; 0020:Axis 1  Positioning  start
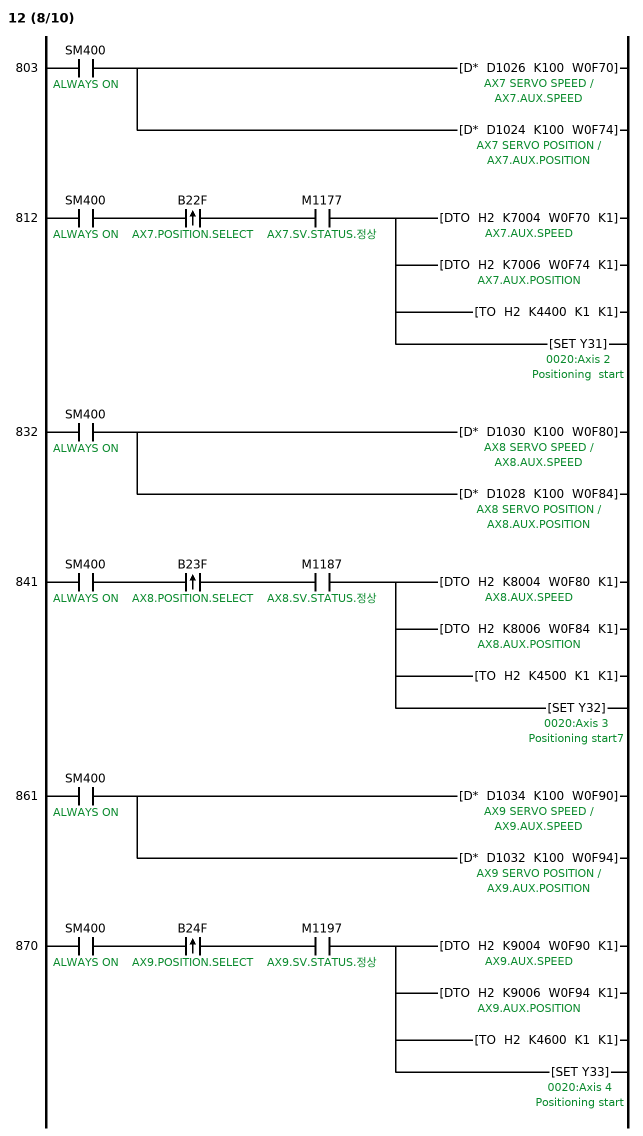
803   LD      SM400  ; ALWAYS ON
      D*      D1026 K100 W0F70  ; AX7 SERVO SPEED / AX7.AUX.SPEED
      D*      D1024 K100 W0F74  ; AX7 SERVO POSITION / AX7.AUX.POSITION
812   LD      SM400  ; ALWAYS ON
      ANDP    B22F  ; AX7.POSITION.SELECT
      AND     M1177  ; AX7.SV.STATUS.정상
      DTO     H2 K7004 W0F70 K1
      DTO     H2 K7006 W0F74 K1
      TO      H2 K4400 K1 K1
      SET     Y31  ; 0020:Axis 2  Positioning  start
832   LD      SM400  ; ALWAYS ON
      D*      D1030 K100 W0F80  ; AX8 SERVO SPEED / AX8.AUX.SPEED
      D*      D1028 K100 W0F84  ; AX8 SERVO POSITION / AX8.AUX.POSITION
841   LD      SM400  ; ALWAYS ON
      ANDP    B23F  ; AX8.POSITION.SELECT
      AND     M1187  ; AX8.SV.STATUS.정상
      DTO     H2 K8004 W0F80 K1
      DTO     H2 K8006 W0F84 K1
      TO      H2 K4500 K1 K1
      SET     Y32  ; 0020:Axis 3 Positioning start7
861   LD      SM400  ; ALWAYS ON
      D*      D1034 K100 W0F90  ; AX9 SERVO SPEED / AX9.AUX.SPEED
      D*      D1032 K100 W0F94  ; AX9 SERVO POSITION / AX9.AUX.POSITION
870   LD      SM400  ; ALWAYS ON
      ANDP    B24F  ; AX9.POSITION.SELECT
      AND     M1197  ; AX9.SV.STATUS.정상
      DTO     H2 K9004 W0F90 K1
      DTO     H2 K9006 W0F94 K1
      TO      H2 K4600 K1 K1
      SET     Y33  ; 0020:Axis 4 Positioning start
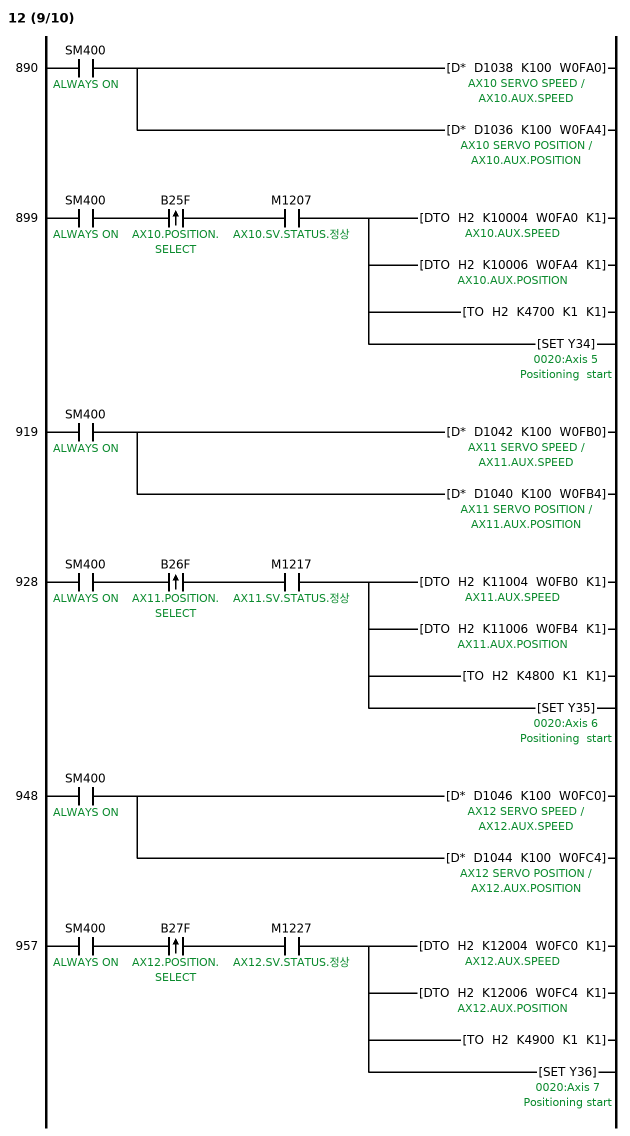
890   LD      SM400  ; ALWAYS ON
      D*      D1038 K100 W0FA0  ; AX10 SERVO SPEED / AX10.AUX.SPEED
      D*      D1036 K100 W0FA4  ; AX10 SERVO POSITION / AX10.AUX.POSITION
899   LD      SM400  ; ALWAYS ON
      ANDP    B25F  ; AX10.POSITION.SELECT
      AND     M1207  ; AX10.SV.STATUS.정상
      DTO     H2 K10004 W0FA0 K1
      DTO     H2 K10006 W0FA4 K1
      TO      H2 K4700 K1 K1
      SET     Y34  ; 0020:Axis 5  Positioning  start
919   LD      SM400  ; ALWAYS ON
      D*      D1042 K100 W0FB0  ; AX11 SERVO SPEED / AX11.AUX.SPEED
      D*      D1040 K100 W0FB4  ; AX11 SERVO POSITION / AX11.AUX.POSITION
928   LD      SM400  ; ALWAYS ON
      ANDP    B26F  ; AX11.POSITION.SELECT
      AND     M1217  ; AX11.SV.STATUS.정상
      DTO     H2 K11004 W0FB0 K1
      DTO     H2 K11006 W0FB4 K1
      TO      H2 K4800 K1 K1
      SET     Y35  ; 0020:Axis 6  Positioning  start
948   LD      SM400  ; ALWAYS ON
      D*      D1046 K100 W0FC0  ; AX12 SERVO SPEED / AX12.AUX.SPEED
      D*      D1044 K100 W0FC4  ; AX12 SERVO POSITION / AX12.AUX.POSITION
957   LD      SM400  ; ALWAYS ON
      ANDP    B27F  ; AX12.POSITION.SELECT
      AND     M1227  ; AX12.SV.STATUS.정상
      DTO     H2 K12004 W0FC0 K1
      DTO     H2 K12006 W0FC4 K1
      TO      H2 K4900 K1 K1
      SET     Y36  ; 0020:Axis 7 Positioning start
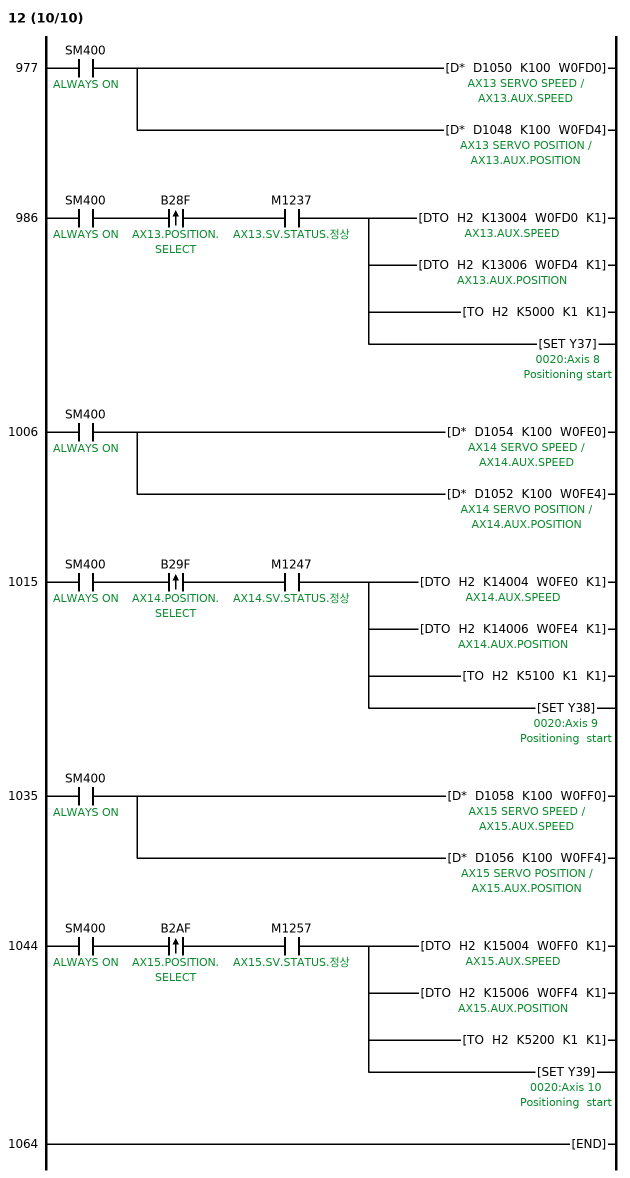
977   LD      SM400  ; ALWAYS ON
      D*      D1050 K100 W0FD0  ; AX13 SERVO SPEED / AX13.AUX.SPEED
      D*      D1048 K100 W0FD4  ; AX13 SERVO POSITION / AX13.AUX.POSITION
986   LD      SM400  ; ALWAYS ON
      ANDP    B28F  ; AX13.POSITION.SELECT
      AND     M1237  ; AX13.SV.STATUS.정상
      DTO     H2 K13004 W0FD0 K1
      DTO     H2 K13006 W0FD4 K1
      TO      H2 K5000 K1 K1
      SET     Y37  ; 0020:Axis 8 Positioning start
1006  LD      SM400  ; ALWAYS ON
      D*      D1054 K100 W0FE0  ; AX14 SERVO SPEED / AX14.AUX.SPEED
      D*      D1052 K100 W0FE4  ; AX14 SERVO POSITION / AX14.AUX.POSITION
1015  LD      SM400  ; ALWAYS ON
      ANDP    B29F  ; AX14.POSITION.SELECT
      AND     M1247  ; AX14.SV.STATUS.정상
      DTO     H2 K14004 W0FE0 K1
      DTO     H2 K14006 W0FE4 K1
      TO      H2 K5100 K1 K1
      SET     Y38  ; 0020:Axis 9  Positioning  start
1035  LD      SM400  ; ALWAYS ON
      D*      D1058 K100 W0FF0  ; AX15 SERVO SPEED / AX15.AUX.SPEED
      D*      D1056 K100 W0FF4  ; AX15 SERVO POSITION / AX15.AUX.POSITION
1044  LD      SM400  ; ALWAYS ON
      ANDP    B2AF  ; AX15.POSITION.SELECT
      AND     M1257  ; AX15.SV.STATUS.정상
      DTO     H2 K15004 W0FF0 K1
      DTO     H2 K15006 W0FF4 K1
      TO      H2 K5200 K1 K1
      SET     Y39  ; 0020:Axis 10  Positioning  start
1064  END
END_PROGRAM

PROGRAM 06  // ALARM
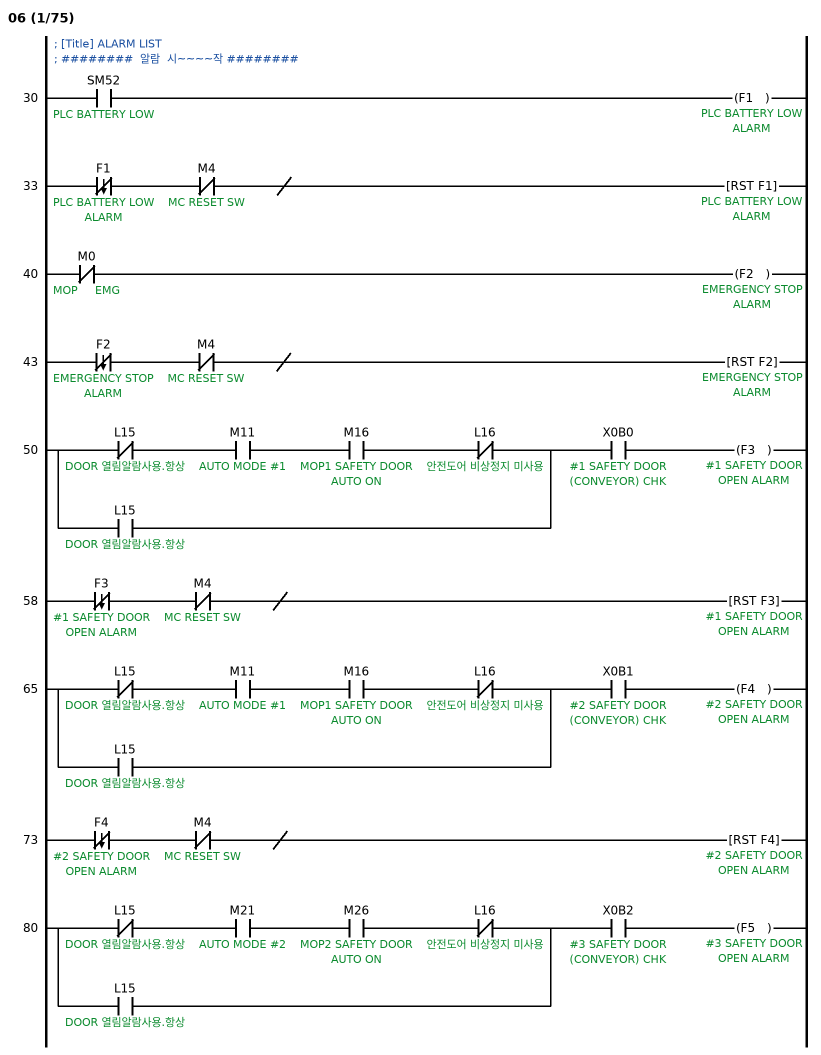
; [Title] ALARM LIST
; ########  알람  시~~~~작 ########
30    LD      SM52  ; PLC BATTERY LOW
      OUT     F1  ; PLC BATTERY LOW ALARM
33    LDFI    F1  ; PLC BATTERY LOW ALARM
      ANI     M4  ; MC RESET SW
      INV
      RST     F1  ; PLC BATTERY LOW ALARM
40    LDI     M0  ; MOP     EMG
      OUT     F2  ; EMERGENCY STOP ALARM
43    LDFI    F2  ; EMERGENCY STOP ALARM
      ANI     M4  ; MC RESET SW
      INV
      RST     F2  ; EMERGENCY STOP ALARM
50    LDI     L15  ; DOOR 열림알람사용.항상
      AND     M11  ; AUTO MODE #1
      AND     M16  ; MOP1 SAFETY DOOR AUTO ON
      ANI     L16  ; 안전도어 비상정지 미사용
      OR      L15  ; DOOR 열림알람사용.항상
      AND     X0B0  ; #1 SAFETY DOOR (CONVEYOR) CHK
      OUT     F3  ; #1 SAFETY DOOR  OPEN ALARM
58    LDFI    F3  ; #1 SAFETY DOOR  OPEN ALARM
      ANI     M4  ; MC RESET SW
      INV
      RST     F3  ; #1 SAFETY DOOR  OPEN ALARM
65    LDI     L15  ; DOOR 열림알람사용.항상
      AND     M11  ; AUTO MODE #1
      AND     M16  ; MOP1 SAFETY DOOR AUTO ON
      ANI     L16  ; 안전도어 비상정지 미사용
      OR      L15  ; DOOR 열림알람사용.항상
      AND     X0B1  ; #2 SAFETY DOOR (CONVEYOR) CHK
      OUT     F4  ; #2 SAFETY DOOR  OPEN ALARM
73    LDFI    F4  ; #2 SAFETY DOOR  OPEN ALARM
      ANI     M4  ; MC RESET SW
      INV
      RST     F4  ; #2 SAFETY DOOR  OPEN ALARM
80    LDI     L15  ; DOOR 열림알람사용.항상
      AND     M21  ; AUTO MODE #2
      AND     M26  ; MOP2 SAFETY DOOR AUTO ON
      ANI     L16  ; 안전도어 비상정지 미사용
      OR      L15  ; DOOR 열림알람사용.항상
      AND     X0B2  ; #3 SAFETY DOOR (CONVEYOR) CHK
      OUT     F5  ; #3 SAFETY DOOR  OPEN ALARM
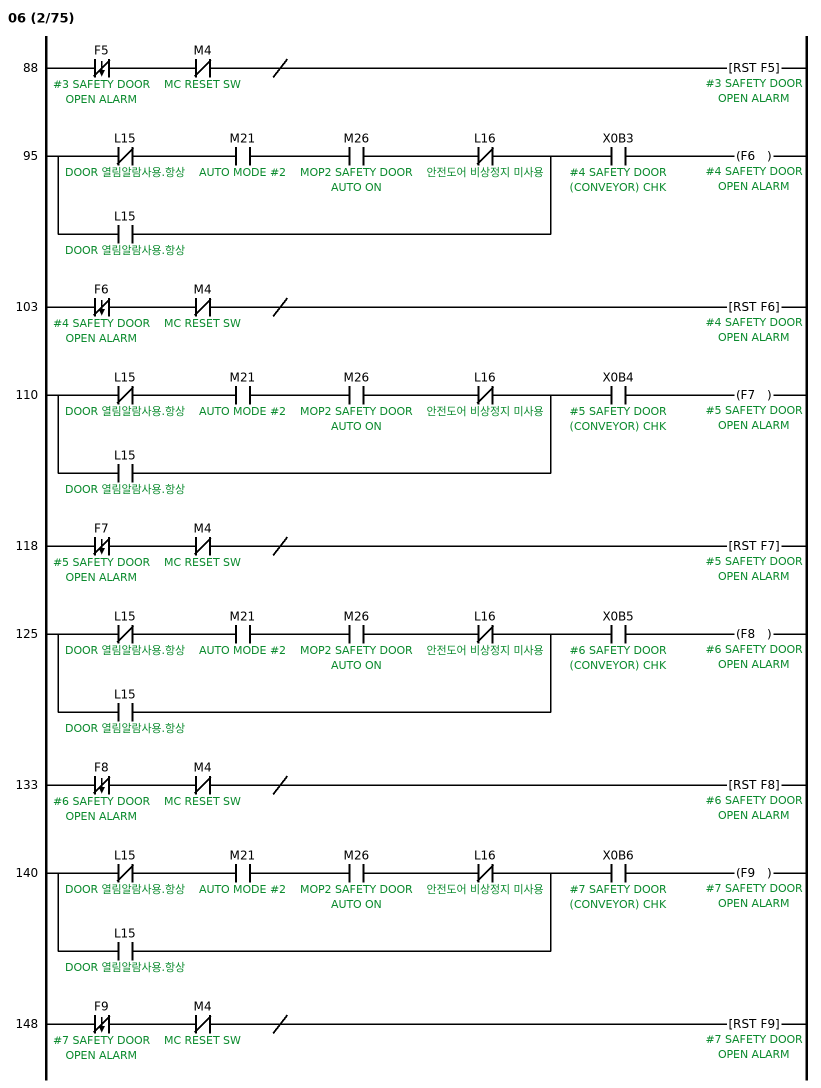
88    LDFI    F5  ; #3 SAFETY DOOR  OPEN ALARM
      ANI     M4  ; MC RESET SW
      INV
      RST     F5  ; #3 SAFETY DOOR  OPEN ALARM
95    LDI     L15  ; DOOR 열림알람사용.항상
      AND     M21  ; AUTO MODE #2
      AND     M26  ; MOP2 SAFETY DOOR AUTO ON
      ANI     L16  ; 안전도어 비상정지 미사용
      OR      L15  ; DOOR 열림알람사용.항상
      AND     X0B3  ; #4 SAFETY DOOR (CONVEYOR) CHK
      OUT     F6  ; #4 SAFETY DOOR  OPEN ALARM
103   LDFI    F6  ; #4 SAFETY DOOR  OPEN ALARM
      ANI     M4  ; MC RESET SW
      INV
      RST     F6  ; #4 SAFETY DOOR  OPEN ALARM
110   LDI     L15  ; DOOR 열림알람사용.항상
      AND     M21  ; AUTO MODE #2
      AND     M26  ; MOP2 SAFETY DOOR AUTO ON
      ANI     L16  ; 안전도어 비상정지 미사용
      OR      L15  ; DOOR 열림알람사용.항상
      AND     X0B4  ; #5 SAFETY DOOR (CONVEYOR) CHK
      OUT     F7  ; #5 SAFETY DOOR  OPEN ALARM
118   LDFI    F7  ; #5 SAFETY DOOR  OPEN ALARM
      ANI     M4  ; MC RESET SW
      INV
      RST     F7  ; #5 SAFETY DOOR  OPEN ALARM
125   LDI     L15  ; DOOR 열림알람사용.항상
      AND     M21  ; AUTO MODE #2
      AND     M26  ; MOP2 SAFETY DOOR AUTO ON
      ANI     L16  ; 안전도어 비상정지 미사용
      OR      L15  ; DOOR 열림알람사용.항상
      AND     X0B5  ; #6 SAFETY DOOR (CONVEYOR) CHK
      OUT     F8  ; #6 SAFETY DOOR  OPEN ALARM
133   LDFI    F8  ; #6 SAFETY DOOR  OPEN ALARM
      ANI     M4  ; MC RESET SW
      INV
      RST     F8  ; #6 SAFETY DOOR  OPEN ALARM
140   LDI     L15  ; DOOR 열림알람사용.항상
      AND     M21  ; AUTO MODE #2
      AND     M26  ; MOP2 SAFETY DOOR AUTO ON
      ANI     L16  ; 안전도어 비상정지 미사용
      OR      L15  ; DOOR 열림알람사용.항상
      AND     X0B6  ; #7 SAFETY DOOR (CONVEYOR) CHK
      OUT     F9  ; #7 SAFETY DOOR  OPEN ALARM
148   LDFI    F9  ; #7 SAFETY DOOR  OPEN ALARM
      ANI     M4  ; MC RESET SW
      INV
      RST     F9  ; #7 SAFETY DOOR  OPEN ALARM
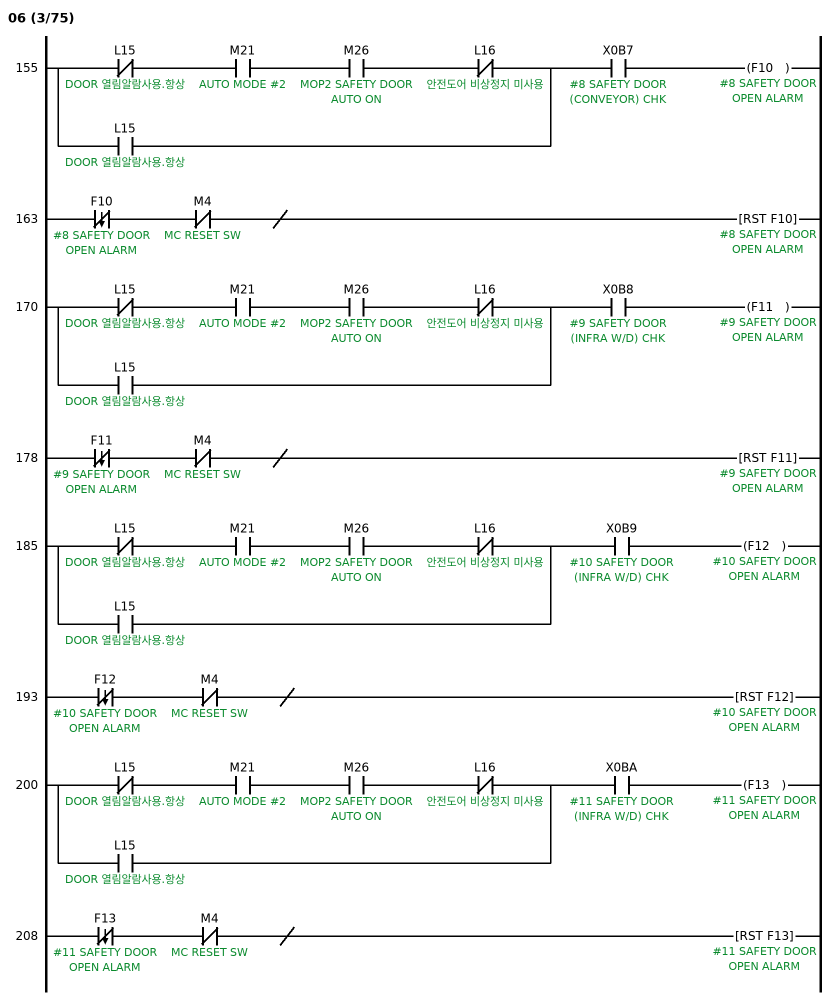
155   LDI     L15  ; DOOR 열림알람사용.항상
      AND     M21  ; AUTO MODE #2
      AND     M26  ; MOP2 SAFETY DOOR AUTO ON
      ANI     L16  ; 안전도어 비상정지 미사용
      OR      L15  ; DOOR 열림알람사용.항상
      AND     X0B7  ; #8 SAFETY DOOR (CONVEYOR) CHK
      OUT     F10  ; #8 SAFETY DOOR  OPEN ALARM
163   LDFI    F10  ; #8 SAFETY DOOR  OPEN ALARM
      ANI     M4  ; MC RESET SW
      INV
      RST     F10  ; #8 SAFETY DOOR  OPEN ALARM
170   LDI     L15  ; DOOR 열림알람사용.항상
      AND     M21  ; AUTO MODE #2
      AND     M26  ; MOP2 SAFETY DOOR AUTO ON
      ANI     L16  ; 안전도어 비상정지 미사용
      OR      L15  ; DOOR 열림알람사용.항상
      AND     X0B8  ; #9 SAFETY DOOR (INFRA W/D) CHK
      OUT     F11  ; #9 SAFETY DOOR  OPEN ALARM
178   LDFI    F11  ; #9 SAFETY DOOR  OPEN ALARM
      ANI     M4  ; MC RESET SW
      INV
      RST     F11  ; #9 SAFETY DOOR  OPEN ALARM
185   LDI     L15  ; DOOR 열림알람사용.항상
      AND     M21  ; AUTO MODE #2
      AND     M26  ; MOP2 SAFETY DOOR AUTO ON
      ANI     L16  ; 안전도어 비상정지 미사용
      OR      L15  ; DOOR 열림알람사용.항상
      AND     X0B9  ; #10 SAFETY DOOR (INFRA W/D) CHK
      OUT     F12  ; #10 SAFETY DOOR OPEN ALARM
193   LDFI    F12  ; #10 SAFETY DOOR OPEN ALARM
      ANI     M4  ; MC RESET SW
      INV
      RST     F12  ; #10 SAFETY DOOR OPEN ALARM
200   LDI     L15  ; DOOR 열림알람사용.항상
      AND     M21  ; AUTO MODE #2
      AND     M26  ; MOP2 SAFETY DOOR AUTO ON
      ANI     L16  ; 안전도어 비상정지 미사용
      OR      L15  ; DOOR 열림알람사용.항상
      AND     X0BA  ; #11 SAFETY DOOR (INFRA W/D) CHK
      OUT     F13  ; #11 SAFETY DOOR OPEN ALARM
208   LDFI    F13  ; #11 SAFETY DOOR OPEN ALARM
      ANI     M4  ; MC RESET SW
      INV
      RST     F13  ; #11 SAFETY DOOR OPEN ALARM
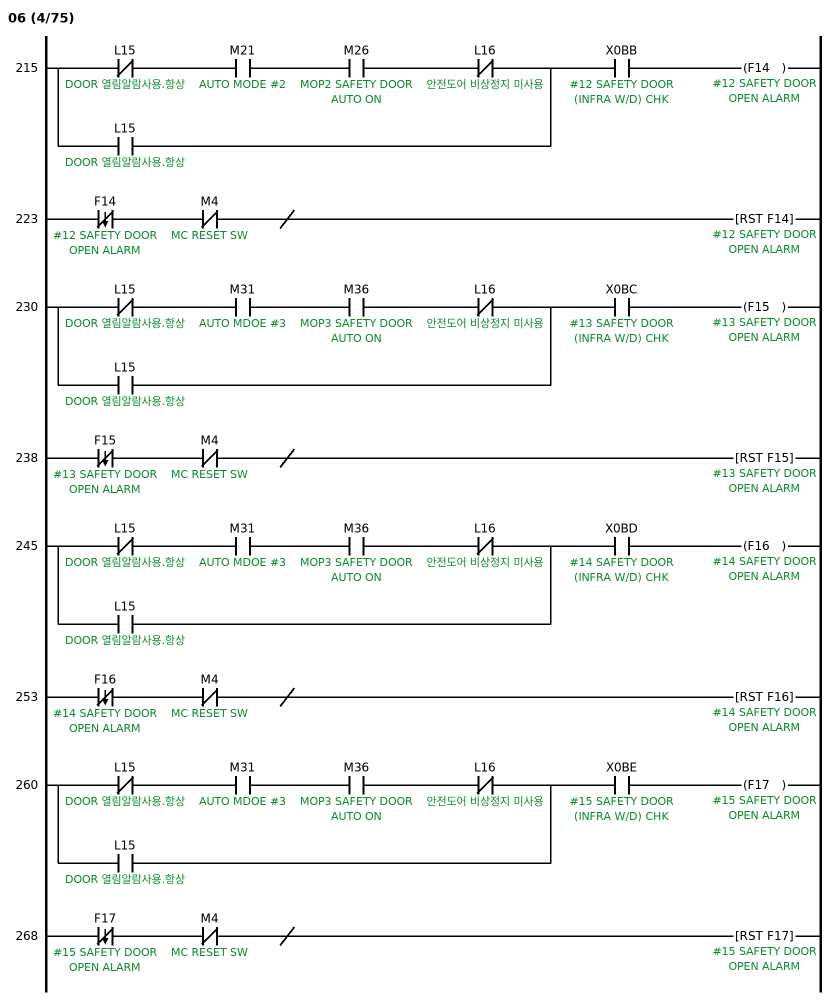
215   LDI     L15  ; DOOR 열림알람사용.항상
      AND     M21  ; AUTO MODE #2
      AND     M26  ; MOP2 SAFETY DOOR AUTO ON
      ANI     L16  ; 안전도어 비상정지 미사용
      OR      L15  ; DOOR 열림알람사용.항상
      AND     X0BB  ; #12 SAFETY DOOR (INFRA W/D) CHK
      OUT     F14  ; #12 SAFETY DOOR OPEN ALARM
223   LDFI    F14  ; #12 SAFETY DOOR OPEN ALARM
      ANI     M4  ; MC RESET SW
      INV
      RST     F14  ; #12 SAFETY DOOR OPEN ALARM
230   LDI     L15  ; DOOR 열림알람사용.항상
      AND     M31  ; AUTO MDOE #3
      AND     M36  ; MOP3 SAFETY DOOR AUTO ON
      ANI     L16  ; 안전도어 비상정지 미사용
      OR      L15  ; DOOR 열림알람사용.항상
      AND     X0BC  ; #13 SAFETY DOOR (INFRA W/D) CHK
      OUT     F15  ; #13 SAFETY DOOR OPEN ALARM
238   LDFI    F15  ; #13 SAFETY DOOR OPEN ALARM
      ANI     M4  ; MC RESET SW
      INV
      RST     F15  ; #13 SAFETY DOOR OPEN ALARM
245   LDI     L15  ; DOOR 열림알람사용.항상
      AND     M31  ; AUTO MDOE #3
      AND     M36  ; MOP3 SAFETY DOOR AUTO ON
      ANI     L16  ; 안전도어 비상정지 미사용
      OR      L15  ; DOOR 열림알람사용.항상
      AND     X0BD  ; #14 SAFETY DOOR (INFRA W/D) CHK
      OUT     F16  ; #14 SAFETY DOOR OPEN ALARM
253   LDFI    F16  ; #14 SAFETY DOOR OPEN ALARM
      ANI     M4  ; MC RESET SW
      INV
      RST     F16  ; #14 SAFETY DOOR OPEN ALARM
260   LDI     L15  ; DOOR 열림알람사용.항상
      AND     M31  ; AUTO MDOE #3
      AND     M36  ; MOP3 SAFETY DOOR AUTO ON
      ANI     L16  ; 안전도어 비상정지 미사용
      OR      L15  ; DOOR 열림알람사용.항상
      AND     X0BE  ; #15 SAFETY DOOR (INFRA W/D) CHK
      OUT     F17  ; #15 SAFETY DOOR OPEN ALARM
268   LDFI    F17  ; #15 SAFETY DOOR OPEN ALARM
      ANI     M4  ; MC RESET SW
      INV
      RST     F17  ; #15 SAFETY DOOR OPEN ALARM
